KUKA KRL program: EPS_2_25999_MH2A_A_20251114084354.src

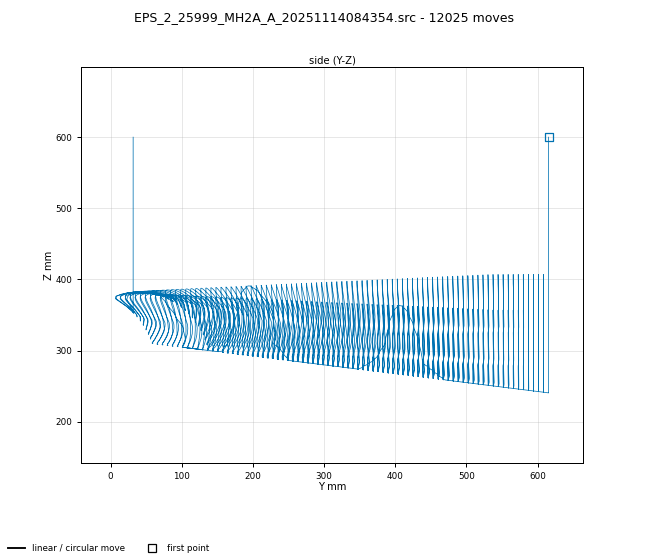
[picture p0: tool path of EPS_2_25999_MH2A_A_20251114084354.src, 12025 of 12027 moves have a stored position in this frame; points joined in program order, loops and branches not executed]
&ACCESS RVP
&REL 4
&COMMENT QRS 19112012
&PARAM EDITMASK = *
DEF PART()
EXT BAS (BAS_COMMAND :IN,REAL :IN )
INT I
BAS (#INITMOV,0 )

;KUKA QRS Post kuka4.cps  Date:22-06-2017 !

File_ID=2913

QRS_PRE_INIT()

;Init var - Until changes are made in qrs_pre_init
Outlet_Square_prg=0
Inlet_1_Square_prg=0
Inlet_2_Square_prg=0
Inlet_3_Square_prg=0
Inlet_4_Square_prg=0
Inlet_5_Square_prg=0

Outlet_1={X 0.000, Y 536.360, Z 332.000, B 0.000, E1 0.000 }
Inlet_1={X 0.000, Y 539.940, Z 282.000, B 0.000, E1 194.000 }
Outlet_1_type=150
Inlet_1_type=150
;QRS#1=Sidecore dimensions
;QRS#2=150-6" PVC SDR 28
;QRS#3=150-6" PVC SDR 28
;QRS#4=
;QRS#5=
;QRS#6=
;QRS#7=
;QRS#8=
;QRS#9=10-06 PSX
;QRS#10=10-06 PSX
;QRS#11=
;QRS#12=
;QRS#13=
;QRS#14=
;QRS#15=
;QRS#16=1220x127x686 2,25'
;QRS#17=EPS Height
;QRS#18=407
;QRS#19=*
;QRS#20= UPDATED VERSION 22-06-2017
;QRS#21=*
Outlet_Square=070
Inlet_1_Square=070
Inlet_2_Square=0
Inlet_3_Square=0
Inlet_4_Square=0
Inlet_5_Square=0
Mill_Square=1
Outlet_Square_Prg=203
Inlet_1_Square_prg=203

QRS_INIT()

$ADVANCE=5

; T1
PTP {E1 173.62,E2 173.62}
PTP {X 0,Y 615.486,A -85,B 0,C 180,E1 173.62,E2 173.62,E3 0,E4 0,E5 0,E6 0}
QRS_SPEED_INIT()
LIN {X 0,Y 615.486,Z 600,A -85,B 0,C 180,E1 173.62,E2 173.62,E3 0,E4 0,E5 0,E6 0} C_VEL
LIN {X 0,Y 615.486,Z 250.689,A -85,B 0,C 180,E1 173.62,E2 173.62} C_VEL
LIN {X 0,Y 615.486,Z 242.512,A -85,B 0,C 180,E1 173.62,E2 173.62} C_VEL
LIN {X 0,Y 615.477,Z 240.512,A -85,B 0,C 180,E1 173.434,E2 173.434} C_VEL
LIN {X 0,Y 615.498,Z 240.51,A -85,B 0,C 180,E1 170.803,E2 170.803} C_VEL
LIN {X 0,Y 615.487,Z 240.512,A -85,B 0,C 180,E1 168.141,E2 168.141} C_VEL
LIN {X 0,Y 615.477,Z 240.512,A -85,B 0,C 180,E1 165.452,E2 165.452} C_VEL
LIN {X 0,Y 615.487,Z 240.513,A -85,B 0,C 180,E1 162.731,E2 162.731} C_VEL
LIN {X 0,Y 615.49,Z 240.512,A -85,B 0,C 180,E1 159.969,E2 159.969} C_VEL
LIN {X 0,Y 615.493,Z 240.509,A -85,B 0,C 180,E1 157.157,E2 157.157} C_VEL
LIN {X 0,Y 615.478,Z 240.513,A -85,B 0,C 180,E1 154.434,E2 154.434} C_VEL
LIN {X 0,Y 615.479,Z 240.512,A -85,B 0,C 180,E1 152.086,E2 152.086} C_VEL
LIN {X 0,Y 615.49,Z 240.513,A -85,B 0,C 180,E1 149.842,E2 149.842} C_VEL
LIN {X 0,Y 615.495,Z 240.511,A -85,B 0,C 180,E1 147.545,E2 147.545} C_VEL
LIN {X 0,Y 615.487,Z 240.51,A -85,B 0,C 180,E1 145.187,E2 145.187} C_VEL
LIN {X 0,Y 615.487,Z 240.513,A -85,B 0,C 180,E1 142.76,E2 142.76} C_VEL
LIN {X 0,Y 615.479,Z 240.513,A -85,B 0,C 180,E1 139.913,E2 139.913} C_VEL
LIN {X 0,Y 615.5,Z 240.511,A -85,B 0,C 180,E1 137.651,E2 137.651} C_VEL
LIN {X 0,Y 615.477,Z 240.513,A -85,B 0,C 180,E1 134.933,E2 134.933} C_VEL
LIN {X 0,Y 615.49,Z 240.51,A -85,B 0,C 180,E1 132.083,E2 132.083} C_VEL
LIN {X 0,Y 615.491,Z 240.51,A -85,B 0,C 180,E1 129.751,E2 129.751} C_VEL
LIN {X 0,Y 615.476,Z 240.512,A -85,B 0,C 180,E1 126.939,E2 126.939} C_VEL
LIN {X 0,Y 615.481,Z 240.513,A -85,B 0,C 180,E1 124.704,E2 124.704} C_VEL
LIN {X 0,Y 615.498,Z 240.511,A -85,B 0,C 180,E1 122.336,E2 122.336} C_VEL
LIN {X 0,Y 615.49,Z 240.514,A -85,B 0,C 180,E1 119.407,E2 119.407} C_VEL
LIN {X 0,Y 615.492,Z 240.512,A -85,B 0,C 180,E1 116.445,E2 116.445} C_VEL
LIN {X 0,Y 615.483,Z 240.512,A -85,B 0,C 180,E1 113.557,E2 113.557} C_VEL
LIN {X 0,Y 615.485,Z 240.511,A -85,B 0,C 180,E1 110.732,E2 110.732} C_VEL
LIN {X 0,Y 615.492,Z 240.509,A -85,B 0,C 180,E1 108.613,E2 108.613} C_VEL
LIN {X 0,Y 615.483,Z 242.217,A -85,B 0,C 180,E1 107.271,E2 107.271} C_VEL
LIN {X 0,Y 615.491,Z 246.275,A -85,B 0,C 180,E1 104.55,E2 104.55} C_VEL
LIN {X 0,Y 615.487,Z 250.425,A -85,B 0,C 180,E1 101.862,E2 101.862} C_VEL
LIN {X 0,Y 615.47,Z 254.646,A -85,B 0,C 180,E1 99.2,E2 99.2} C_VEL
LIN {X 0,Y 615.491,Z 258.931,A -85,B 0,C 180,E1 96.557,E2 96.557} C_VEL
LIN {X 0,Y 615.464,Z 263.25,A -85,B 0,C 180,E1 93.929,E2 93.929} C_VEL
LIN {X 0,Y 615.465,Z 267.63,A -85,B 0,C 180,E1 91.309,E2 91.309} C_VEL
LIN {X 0,Y 615.493,Z 272.05,A -85,B 0,C 180,E1 88.692,E2 88.692} C_VEL
LIN {X 0,Y 615.433,Z 276.534,A -85,B 0,C 180,E1 86.072,E2 86.072} C_VEL
LIN {X 0,Y 615.492,Z 278.219,A -85,B 0,C 180,E1 85.088,E2 85.088} C_VEL
LIN {X 0,Y 615.471,Z 289.997,A -85,B 0,C 180,E1 84.76,E2 84.76} C_VEL
LIN {X 0,Y 615.441,Z 298.609,A -85,B 0,C 180,E1 84.431,E2 84.431} C_VEL
LIN {X 0,Y 615.429,Z 306.992,A -85,B 0,C 180,E1 84.02,E2 84.02} C_VEL
LIN {X 0,Y 615.456,Z 315.045,A -85,B 0,C 180,E1 83.526,E2 83.526} C_VEL
LIN {X 0,Y 615.498,Z 322.786,A -85,B 0,C 180,E1 82.944,E2 82.944} C_VEL
LIN {X 0,Y 615.496,Z 331.565,A -85,B 0,C 180,E1 82.125,E2 82.125} C_VEL
LIN {X 0,Y 615.497,Z 338.404,A -85,B 0,C 180,E1 81.299,E2 81.299} C_VEL
LIN {X 0,Y 615.495,Z 343.88,A -85,B 0,C 180,E1 80.471,E2 80.471} C_VEL
LIN {X 0,Y 615.49,Z 347.453,A -85,B 0,C 180,E1 79.807,E2 79.807} C_VEL
LIN {X 0,Y 615.492,Z 351.54,A -85,B 0,C 180,E1 78.808,E2 78.808} C_VEL
LIN {X 0,Y 615.491,Z 353.549,A -85,B 0,C 180,E1 78.14,E2 78.14} C_VEL
LIN {X 0,Y 615.496,Z 355.036,A -85,B 0,C 180,E1 77.471,E2 77.471} C_VEL
LIN {X 0,Y 615.491,Z 355.978,A -85,B 0,C 180,E1 76.8,E2 76.8} C_VEL
LIN {X 0,Y 615.491,Z 356.365,A -85,B 0,C 180,E1 76.056,E2 76.056} C_VEL
LIN {X 0,Y 615.493,Z 356.174,A -85,B 0,C 180,E1 75.452,E2 75.452} C_VEL
LIN {X 0,Y 615.491,Z 355.513,A -85,B 0,C 180,E1 74.775,E2 74.775} C_VEL
LIN {X 0,Y 615.491,Z 354.339,A -85,B 0,C 180,E1 74.096,E2 74.096} C_VEL
LIN {X 0,Y 615.492,Z 352.622,A -85,B 0,C 180,E1 73.415,E2 73.415} C_VEL
LIN {X 0,Y 615.496,Z 348.756,A -85,B 0,C 180,E1 72.388,E2 72.388} C_VEL
LIN {X 0,Y 615.496,Z 343.394,A -85,B 0,C 180,E1 71.355,E2 71.355} C_VEL
LIN {X 0,Y 615.498,Z 337.543,A -85,B 0,C 180,E1 70.49,E2 70.49} C_VEL
LIN {X 0,Y 615.496,Z 330.756,A -85,B 0,C 180,E1 69.702,E2 69.702} C_VEL
LIN {X 0,Y 615.497,Z 323.297,A -85,B 0,C 180,E1 69.008,E2 69.008} C_VEL
LIN {X 0,Y 615.471,Z 316.464,A -85,B 0,C 180,E1 68.481,E2 68.481} C_VEL
LIN {X 0,Y 615.468,Z 308.08,A -85,B 0,C 180,E1 67.952,E2 67.952} C_VEL
LIN {X 0,Y 615.494,Z 299.6,A -85,B 0,C 180,E1 67.525,E2 67.525} C_VEL
LIN {X 0,Y 615.487,Z 291.944,A -85,B 0,C 180,E1 67.218,E2 67.218} C_VEL
LIN {X 0,Y 615.496,Z 282.553,A -85,B 0,C 180,E1 66.935,E2 66.935} C_VEL
LIN {X 0,Y 615.485,Z 278.224,A -85,B 0,C 180,E1 66.823,E2 66.823} C_VEL
LIN {X 0,Y 615.458,Z 273.873,A -85,B 0,C 180,E1 64.284,E2 64.284} C_VEL
LIN {X 0,Y 615.494,Z 269.211,A -85,B 0,C 180,E1 61.544,E2 61.544} C_VEL
LIN {X 0,Y 615.444,Z 264.82,A -85,B 0,C 180,E1 58.916,E2 58.916} C_VEL
LIN {X 0,Y 615.444,Z 260.756,A -85,B 0,C 180,E1 56.468,E2 56.468} C_VEL
LIN {X 0,Y 615.462,Z 256.05,A -85,B 0,C 180,E1 53.575,E2 53.575} C_VEL
LIN {X 0,Y 615.42,Z 251.843,A -85,B 0,C 180,E1 50.942,E2 50.942} C_VEL
LIN {X 0,Y 615.456,Z 248.051,A -85,B 0,C 180,E1 48.525,E2 48.525} C_VEL
LIN {X 0,Y 615.495,Z 244.035,A -85,B 0,C 180,E1 45.853,E2 45.853} C_VEL
LIN {X 0,Y 615.491,Z 241.268,A -85,B 0,C 180,E1 44,E2 44} C_VEL
LIN {X 0,Y 615.457,Z 240.51,A -85,B 0,C 180,E1 43.046,E2 43.046} C_VEL
LIN {X 0,Y 615.484,Z 240.512,A -85,B 0,C 180,E1 40.604,E2 40.604} C_VEL
LIN {X 0,Y 615.473,Z 240.506,A -85,B 0,C 180,E1 38.012,E2 38.012} C_VEL
LIN {X 0,Y 615.489,Z 240.512,A -85,B 0,C 180,E1 35.613,E2 35.613} C_VEL
LIN {X 0,Y 615.446,Z 240.512,A -85,B 0,C 180,E1 33.237,E2 33.237} C_VEL
LIN {X 0,Y 615.491,Z 240.513,A -85,B 0,C 180,E1 30.917,E2 30.917} C_VEL
LIN {X 0,Y 615.481,Z 240.504,A -85,B 0,C 180,E1 28.452,E2 28.452} C_VEL
LIN {X 0,Y 615.454,Z 240.511,A -85,B 0,C 180,E1 25.715,E2 25.715} C_VEL
LIN {X 0,Y 615.488,Z 240.509,A -85,B 0,C 180,E1 22.843,E2 22.843} C_VEL
LIN {X 0,Y 615.484,Z 240.512,A -85,B 0,C 180,E1 20.031,E2 20.031} C_VEL
LIN {X 0,Y 615.472,Z 240.507,A -85,B 0,C 180,E1 17.269,E2 17.269} C_VEL
LIN {X 0,Y 615.448,Z 240.512,A -85,B 0,C 180,E1 14.548,E2 14.548} C_VEL
LIN {X 0,Y 615.49,Z 240.511,A -85,B 0,C 180,E1 11.859,E2 11.859} C_VEL
LIN {X 0,Y 615.498,Z 240.503,A -85,B 0,C 180,E1 9.197,E2 9.197} C_VEL
LIN {X 0,Y 615.443,Z 240.512,A -85,B 0,C 180,E1 6.554,E2 6.554} C_VEL
LIN {X 0,Y 615.491,Z 240.511,A -85,B 0,C 180,E1 3.927,E2 3.927} C_VEL
LIN {X 0,Y 615.494,Z 240.504,A -85,B 0,C 180,E1 1.307,E2 1.307} C_VEL
LIN {X 0,Y 615.445,Z 240.512,A -85,B 0,C 180,E1 -1.31,E2 -1.31} C_VEL
LIN {X 0,Y 615.489,Z 240.513,A -85,B 0,C 180,E1 -3.93,E2 -3.93} C_VEL
LIN {X 0,Y 615.489,Z 240.504,A -85,B 0,C 180,E1 -6.591,E2 -6.591} C_VEL
LIN {X 0,Y 615.446,Z 240.513,A -85,B 0,C 180,E1 -9.2,E2 -9.2} C_VEL
LIN {X 0,Y 615.49,Z 240.513,A -85,B 0,C 180,E1 -11.862,E2 -11.862} C_VEL
LIN {X 0,Y 615.483,Z 240.506,A -85,B 0,C 180,E1 -14.55,E2 -14.55} C_VEL
LIN {X 0,Y 615.451,Z 240.511,A -85,B 0,C 180,E1 -17.272,E2 -17.272} C_VEL
LIN {X 0,Y 615.485,Z 240.507,A -85,B 0,C 180,E1 -20.034,E2 -20.034} C_VEL
LIN {X 0,Y 615.487,Z 240.515,A -85,B 0,C 180,E1 -22.845,E2 -22.845} C_VEL
LIN {X 0,Y 615.492,Z 240.506,A -85,B 0,C 180,E1 -25.716,E2 -25.716} C_VEL
LIN {X 0,Y 615.452,Z 240.511,A -85,B 0,C 180,E1 -28.66,E2 -28.66} C_VEL
LIN {X 0,Y 615.486,Z 240.508,A -85,B 0,C 180,E1 -31.088,E2 -31.088} C_VEL
LIN {X 0,Y 615.495,Z 240.503,A -85,B 0,C 180,E1 -33.537,E2 -33.537} C_VEL
LIN {X 0,Y 615.442,Z 240.513,A -85,B 0,C 180,E1 -36.428,E2 -36.428} C_VEL
LIN {X 0,Y 615.489,Z 240.506,A -85,B 0,C 180,E1 -39.064,E2 -39.064} C_VEL
LIN {X 0,Y 615.491,Z 240.505,A -85,B 0,C 180,E1 -41.474,E2 -41.474} C_VEL
LIN {X 0,Y 615.443,Z 240.512,A -85,B 0,C 180,E1 -44.154,E2 -44.154} C_VEL
LIN {X 0,Y 615.492,Z 240.506,A -85,B 0,C 180,E1 -46.953,E2 -46.953} C_VEL
LIN {X 0,Y 615.489,Z 240.512,A -85,B 0,C 180,E1 -49.911,E2 -49.911} C_VEL
LIN {X 0,Y 615.473,Z 240.513,A -85,B 0,C 180,E1 -52.758,E2 -52.758} C_VEL
LIN {X 0,Y 615.474,Z 240.505,A -85,B 0,C 180,E1 -55.302,E2 -55.302} C_VEL
LIN {X 0,Y 615.486,Z 240.709,A -85,B 0,C 180,E1 -57.447,E2 -57.447} C_VEL
LIN {X 0,Y 615.494,Z 249.851,A -85,B 0,C 180,E1 -60.205,E2 -60.205} C_VEL
LIN {X 0,Y 615.493,Z 259.273,A -85,B 0,C 180,E1 -62.954,E2 -62.954} C_VEL
LIN {X 0,Y 615.447,Z 269.012,A -85,B 0,C 180,E1 -65.727,E2 -65.727} C_VEL
LIN {X 0,Y 615.453,Z 277.921,A -85,B 0,C 180,E1 -68.216,E2 -68.216} C_VEL
LIN {X 0,Y 615.447,Z 288.095,A -85,B 0,C 180,E1 -71.008,E2 -71.008} C_VEL
LIN {X 0,Y 615.45,Z 296.996,A -85,B 0,C 180,E1 -73.413,E2 -73.413} C_VEL
LIN {X 0,Y 615.489,Z 307.146,A -85,B 0,C 180,E1 -76.127,E2 -76.127} C_VEL
LIN {X 0,Y 615.476,Z 317.31,A -85,B 0,C 180,E1 -78.808,E2 -78.808} C_VEL
LIN {X 0,Y 615.485,Z 324.917,A -85,B 0,C 180,E1 -80.802,E2 -80.802} C_VEL
LIN {X 0,Y 615.492,Z 338.188,A -85,B 0,C 180,E1 -81.133,E2 -81.133} C_VEL
LIN {X 0,Y 615.472,Z 347.248,A -85,B 0,C 180,E1 -81.464,E2 -81.464} C_VEL
LIN {X 0,Y 615.475,Z 355.931,A -85,B 0,C 180,E1 -81.877,E2 -81.877} C_VEL
LIN {X 0,Y 615.492,Z 364.211,A -85,B 0,C 180,E1 -82.373,E2 -82.373} C_VEL
LIN {X 0,Y 615.499,Z 371.943,A -85,B 0,C 180,E1 -82.943,E2 -82.943} C_VEL
LIN {X 0,Y 615.498,Z 377.655,A -85,B 0,C 180,E1 -83.444,E2 -83.444} C_VEL
LIN {X 0,Y 615.5,Z 383.929,A -85,B 0,C 180,E1 -84.102,E2 -84.102} C_VEL
LIN {X 0,Y 615.495,Z 389.142,A -85,B 0,C 180,E1 -84.76,E2 -84.76} C_VEL
LIN {X 0,Y 615.495,Z 393.487,A -85,B 0,C 180,E1 -85.416,E2 -85.416} C_VEL
LIN {X 0,Y 615.491,Z 398.607,A -85,B 0,C 180,E1 -86.4,E2 -86.4} C_VEL
LIN {X 0,Y 615.488,Z 401.224,A -85,B 0,C 180,E1 -87.056,E2 -87.056} C_VEL
LIN {X 0,Y 615.499,Z 404.087,A -85,B 0,C 180,E1 -88.038,E2 -88.038} C_VEL
LIN {X 0,Y 615.493,Z 405.331,A -85,B 0,C 180,E1 -88.692,E2 -88.692} C_VEL
LIN {X 0,Y 615.491,Z 406.105,A -85,B 0,C 180,E1 -89.347,E2 -89.347} C_VEL
LIN {X 0,Y 615.491,Z 406.389,A -85,B 0,C 180,E1 -90.001,E2 -90.001} C_VEL
LIN {X 0,Y 615.491,Z 406.104,A -85,B 0,C 180,E1 -90.655,E2 -90.655} C_VEL
LIN {X 0,Y 615.493,Z 405.329,A -85,B 0,C 180,E1 -91.309,E2 -91.309} C_VEL
LIN {X 0,Y 615.499,Z 404.083,A -85,B 0,C 180,E1 -91.964,E2 -91.964} C_VEL
LIN {X 0,Y 615.488,Z 401.218,A -85,B 0,C 180,E1 -92.946,E2 -92.946} C_VEL
LIN {X 0,Y 615.491,Z 398.6,A -85,B 0,C 180,E1 -93.601,E2 -93.601} C_VEL
LIN {X 0,Y 615.495,Z 393.478,A -85,B 0,C 180,E1 -94.585,E2 -94.585} C_VEL
LIN {X 0,Y 615.495,Z 387.962,A -85,B 0,C 180,E1 -95.406,E2 -95.406} C_VEL
LIN {X 0,Y 615.498,Z 381.01,A -85,B 0,C 180,E1 -96.228,E2 -96.228} C_VEL
LIN {X 0,Y 615.498,Z 373.855,A -85,B 0,C 180,E1 -96.901,E2 -96.901} C_VEL
LIN {X 0,Y 615.489,Z 366.61,A -85,B 0,C 180,E1 -97.464,E2 -97.464} C_VEL
LIN {X 0,Y 615.483,Z 358.857,A -85,B 0,C 180,E1 -97.959,E2 -97.959} C_VEL
LIN {X 0,Y 615.469,Z 350.903,A -85,B 0,C 180,E1 -98.372,E2 -98.372} C_VEL
LIN {X 0,Y 615.482,Z 341.736,A -85,B 0,C 180,E1 -98.744,E2 -98.744} C_VEL
LIN {X 0,Y 615.493,Z 333.661,A -85,B 0,C 180,E1 -98.992,E2 -98.992} C_VEL
LIN {X 0,Y 615.485,Z 324.911,A -85,B 0,C 180,E1 -99.2,E2 -99.2} C_VEL
LIN {X 0,Y 615.49,Z 314.759,A -85,B 0,C 180,E1 -101.862,E2 -101.862} C_VEL
LIN {X 0,Y 615.469,Z 304.605,A -85,B 0,C 180,E1 -104.55,E2 -104.55} C_VEL
LIN {X 0,Y 615.472,Z 294.44,A -85,B 0,C 180,E1 -107.272,E2 -107.272} C_VEL
LIN {X 0,Y 615.442,Z 284.276,A -85,B 0,C 180,E1 -110.035,E2 -110.035} C_VEL
LIN {X 0,Y 615.433,Z 275.946,A -85,B 0,C 180,E1 -112.333,E2 -112.333} C_VEL
LIN {X 0,Y 615.495,Z 266.454,A -85,B 0,C 180,E1 -114.992,E2 -114.992} C_VEL
LIN {X 0,Y 615.475,Z 257.545,A -85,B 0,C 180,E1 -117.547,E2 -117.547} C_VEL
LIN {X 0,Y 615.488,Z 248.618,A -85,B 0,C 180,E1 -120.161,E2 -120.161} C_VEL
LIN {X 0,Y 615.485,Z 240.511,A -85,B 0,C 180,E1 -122.652,E2 -122.652} C_VEL
LIN {X 0,Y 615.485,Z 240.511,A -85,B 0,C 180,E1 -124.816,E2 -124.816} C_VEL
LIN {X 0,Y 615.492,Z 240.513,A -85,B 0,C 180,E1 -127.243,E2 -127.243} C_VEL
LIN {X 0,Y 615.48,Z 240.513,A -85,B 0,C 180,E1 -130.088,E2 -130.088} C_VEL
LIN {X 0,Y 615.496,Z 240.513,A -85,B 0,C 180,E1 -132.353,E2 -132.353} C_VEL
LIN {X 0,Y 615.49,Z 240.51,A -85,B 0,C 180,E1 -135.069,E2 -135.069} C_VEL
LIN {X 0,Y 615.476,Z 240.512,A -85,B 0,C 180,E1 -137.922,E2 -137.922} C_VEL
LIN {X 0,Y 615.483,Z 240.512,A -85,B 0,C 180,E1 -140.249,E2 -140.249} C_VEL
LIN {X 0,Y 615.478,Z 240.512,A -85,B 0,C 180,E1 -143.065,E2 -143.065} C_VEL
LIN {X 0,Y 615.48,Z 240.513,A -85,B 0,C 180,E1 -145.301,E2 -145.301} C_VEL
LIN {X 0,Y 615.492,Z 240.512,A -85,B 0,C 180,E1 -147.669,E2 -147.669} C_VEL
LIN {X 0,Y 615.494,Z 240.514,A -85,B 0,C 180,E1 -150.593,E2 -150.593} C_VEL
LIN {X 0,Y 615.477,Z 240.513,A -85,B 0,C 180,E1 -152.958,E2 -152.958} C_VEL
LIN {X 0,Y 615.494,Z 240.513,A -85,B 0,C 180,E1 -155.727,E2 -155.727} C_VEL
LIN {X 0,Y 615.494,Z 240.512,A -85,B 0,C 180,E1 -158.568,E2 -158.568} C_VEL
LIN {X 0,Y 615.479,Z 240.512,A -85,B 0,C 180,E1 -161.399,E2 -161.399} C_VEL
LIN {X 0,Y 615.491,Z 240.51,A -85,B 0,C 180,E1 -164.094,E2 -164.094} C_VEL
LIN {X 0,Y 615.497,Z 240.513,A -85,B 0,C 180,E1 -166.798,E2 -166.798} C_VEL
LIN {X 0,Y 615.477,Z 240.513,A -85,B 0,C 180,E1 -169.472,E2 -169.472} C_VEL
LIN {X 0,Y 615.481,Z 240.512,A -85,B 0,C 180,E1 -172.123,E2 -172.123} C_VEL
LIN {X 0,Y 615.487,Z 240.513,A -85,B 0,C 180,E1 -174.758,E2 -174.758} C_VEL
LIN {X 0,Y 615.491,Z 240.509,A -85,B 0,C 180,E1 -177.381,E2 -177.381} C_VEL
LIN {X 0,Y 615.489,Z 240.514,A -85,B 0,C 180,E1 -179.999,E2 -179.999} C_VEL
LIN {X 0,Y 615.479,Z 240.512,A -85,B 0,C 180,E1 -182.617,E2 -182.617} C_VEL
LIN {X 0,Y 615.497,Z 240.509,A -85,B 0,C 180,E1 -185.24,E2 -185.24} C_VEL
LIN {X 0,Y 615.477,Z 240.512,A -85,B 0,C 180,E1 -186.566,E2 -186.566} C_VEL
LIN {X 0,Y 614.814,Z 240.657,A -85,B 0,C 180,E1 -187.112,E2 -187.112} C_VEL
LIN {X 0,Y 611.991,Z 241.07,A -85,B 0,C 180,E1 -187.998,E2 -187.998} C_VEL
LIN {X 0,Y 609.6,Z 241.378,A -85,B 0,C 180,E1 -188.711,E2 -188.711} C_VEL
LIN {X 0,Y 608.56,Z 241.496,A -85,B 0,C 180,E1 -189.26,E2 -189.26} C_VEL
LIN {X 0,Y 608.468,Z 241.506,A -85,B 0,C 180,E1 -189.447,E2 -189.447} C_VEL
LIN {X 0,Y 608.461,Z 241.509,A -85,B 0,C 180,E1 -191.998,E2 -191.998} C_VEL
LIN {X 0,Y 608.47,Z 241.506,A -85,B 0,C 180,E1 -194.719,E2 -194.719} C_VEL
LIN {X 0,Y 608.453,Z 241.508,A -85,B 0,C 180,E1 -197.475,E2 -197.475} C_VEL
LIN {X 0,Y 608.463,Z 241.508,A -85,B 0,C 180,E1 -200.272,E2 -200.272} C_VEL
LIN {X 0,Y 608.451,Z 241.51,A -85,B 0,C 180,E1 -203.122,E2 -203.122} C_VEL
LIN {X 0,Y 608.463,Z 241.507,A -85,B 0,C 180,E1 -205.718,E2 -205.718} C_VEL
LIN {X 0,Y 608.452,Z 241.511,A -85,B 0,C 180,E1 -208.265,E2 -208.265} C_VEL
LIN {X 0,Y 608.474,Z 241.506,A -85,B 0,C 180,E1 -210.542,E2 -210.542} C_VEL
LIN {X 0,Y 608.462,Z 241.507,A -85,B 0,C 180,E1 -212.877,E2 -212.877} C_VEL
LIN {X 0,Y 608.44,Z 241.512,A -85,B 0,C 180,E1 -215.276,E2 -215.276} C_VEL
LIN {X 0,Y 608.464,Z 241.507,A -85,B 0,C 180,E1 -217.744,E2 -217.744} C_VEL
LIN {X 0,Y 608.447,Z 241.511,A -85,B 0,C 180,E1 -220.328,E2 -220.328} C_VEL
LIN {X 0,Y 608.447,Z 241.509,A -85,B 0,C 180,E1 -222.958,E2 -222.958} C_VEL
LIN {X 0,Y 608.453,Z 241.508,A -85,B 0,C 180,E1 -225.734,E2 -225.734} C_VEL
LIN {X 0,Y 608.462,Z 241.508,A -85,B 0,C 180,E1 -228.655,E2 -228.655} C_VEL
LIN {X 0,Y 608.464,Z 241.508,A -85,B 0,C 180,E1 -231.411,E2 -231.411} C_VEL
LIN {X 0,Y 608.471,Z 241.506,A -85,B 0,C 180,E1 -233.948,E2 -233.948} C_VEL
LIN {X 0,Y 608.472,Z 241.506,A -85,B 0,C 180,E1 -236.329,E2 -236.329} C_VEL
LIN {X 0,Y 608.466,Z 241.508,A -85,B 0,C 180,E1 -238.725,E2 -238.725} C_VEL
LIN {X 0,Y 608.471,Z 241.506,A -85,B 0,C 180,E1 -241.376,E2 -241.376} C_VEL
LIN {X 0,Y 608.444,Z 241.509,A -85,B 0,C 180,E1 -243.964,E2 -243.964} C_VEL
LIN {X 0,Y 608.461,Z 241.507,A -85,B 0,C 180,E1 -246.154,E2 -246.154} C_VEL
LIN {X 0,Y 608.468,Z 241.506,A -85,B 0,C 180,E1 -248.308,E2 -248.308} C_VEL
LIN {X 0,Y 608.467,Z 241.506,A -85,B 0,C 180,E1 -251.278,E2 -251.278} C_VEL
LIN {X 0,Y 608.442,Z 241.748,A -85,B 0,C 180,E1 -251.827,E2 -251.827} C_VEL
LIN {X 0,Y 608.45,Z 245.854,A -85,B 0,C 180,E1 -254.593,E2 -254.593} C_VEL
LIN {X 0,Y 608.451,Z 249.952,A -85,B 0,C 180,E1 -257.322,E2 -257.322} C_VEL
LIN {X 0,Y 608.44,Z 254.187,A -85,B 0,C 180,E1 -260.022,E2 -260.022} C_VEL
LIN {X 0,Y 608.43,Z 258.477,A -85,B 0,C 180,E1 -262.699,E2 -262.699} C_VEL
LIN {X 0,Y 608.455,Z 262.818,A -85,B 0,C 180,E1 -265.362,E2 -265.362} C_VEL
LIN {X 0,Y 608.404,Z 267.215,A -85,B 0,C 180,E1 -268.013,E2 -268.013} C_VEL
LIN {X 0,Y 608.407,Z 271.661,A -85,B 0,C 180,E1 -270.661,E2 -270.661} C_VEL
LIN {X 0,Y 608.41,Z 276.158,A -85,B 0,C 180,E1 -273.31,E2 -273.31} C_VEL
LIN {X 0,Y 608.414,Z 278.71,A -85,B 0,C 180,E1 -274.803,E2 -274.803} C_VEL
LIN {X 0,Y 608.465,Z 290.221,A -85,B 0,C 180,E1 -275.135,E2 -275.135} C_VEL
LIN {X 0,Y 608.452,Z 298.827,A -85,B 0,C 180,E1 -275.467,E2 -275.467} C_VEL
LIN {X 0,Y 608.416,Z 307.241,A -85,B 0,C 180,E1 -275.883,E2 -275.883} C_VEL
LIN {X 0,Y 608.435,Z 314.894,A -85,B 0,C 180,E1 -276.352,E2 -276.352} C_VEL
LIN {X 0,Y 608.467,Z 322.027,A -85,B 0,C 180,E1 -276.882,E2 -276.882} C_VEL
LIN {X 0,Y 608.464,Z 328.587,A -85,B 0,C 180,E1 -277.465,E2 -277.465} C_VEL
LIN {X 0,Y 608.458,Z 334.831,A -85,B 0,C 180,E1 -278.133,E2 -278.133} C_VEL
LIN {X 0,Y 608.448,Z 340.029,A -85,B 0,C 180,E1 -278.803,E2 -278.803} C_VEL
LIN {X 0,Y 608.432,Z 343.398,A -85,B 0,C 180,E1 -279.305,E2 -279.305} C_VEL
LIN {X 0,Y 608.433,Z 347.195,A -85,B 0,C 180,E1 -279.977,E2 -279.977} C_VEL
LIN {X 0,Y 608.424,Z 351.373,A -85,B 0,C 180,E1 -280.946,E2 -280.946} C_VEL
LIN {X 0,Y 608.434,Z 354.534,A -85,B 0,C 180,E1 -281.999,E2 -281.999} C_VEL
LIN {X 0,Y 608.416,Z 355.871,A -85,B 0,C 180,E1 -282.677,E2 -282.677} C_VEL
LIN {X 0,Y 608.433,Z 356.701,A -85,B 0,C 180,E1 -283.356,E2 -283.356} C_VEL
LIN {X 0,Y 608.419,Z 357,A -85,B 0,C 180,E1 -284.038,E2 -284.038} C_VEL
LIN {X 0,Y 608.42,Z 356.707,A -85,B 0,C 180,E1 -284.721,E2 -284.721} C_VEL
LIN {X 0,Y 608.416,Z 355.88,A -85,B 0,C 180,E1 -285.406,E2 -285.406} C_VEL
LIN {X 0,Y 608.447,Z 353.454,A -85,B 0,C 180,E1 -286.531,E2 -286.531} C_VEL
LIN {X 0,Y 608.428,Z 350.112,A -85,B 0,C 180,E1 -287.476,E2 -287.476} C_VEL
LIN {X 0,Y 608.443,Z 345.378,A -85,B 0,C 180,E1 -288.441,E2 -288.441} C_VEL
LIN {X 0,Y 608.464,Z 340.518,A -85,B 0,C 180,E1 -289.218,E2 -289.218} C_VEL
LIN {X 0,Y 608.463,Z 335.138,A -85,B 0,C 180,E1 -289.921,E2 -289.921} C_VEL
LIN {X 0,Y 608.46,Z 329.413,A -85,B 0,C 180,E1 -290.544,E2 -290.544} C_VEL
LIN {X 0,Y 608.47,Z 322.648,A -85,B 0,C 180,E1 -291.157,E2 -291.157} C_VEL
LIN {X 0,Y 608.457,Z 315.575,A -85,B 0,C 180,E1 -291.691,E2 -291.691} C_VEL
LIN {X 0,Y 608.45,Z 308.474,A -85,B 0,C 180,E1 -292.137,E2 -292.137} C_VEL
LIN {X 0,Y 608.503,Z 299.706,A -85,B 0,C 180,E1 -292.582,E2 -292.582} C_VEL
LIN {X 0,Y 608.48,Z 290.597,A -85,B 0,C 180,E1 -292.942,E2 -292.942} C_VEL
LIN {X 0,Y 608.495,Z 281.297,A -85,B 0,C 180,E1 -293.211,E2 -293.211} C_VEL
LIN {X 0,Y 608.426,Z 278.72,A -85,B 0,C 180,E1 -293.281,E2 -293.281} C_VEL
LIN {X 0,Y 608.399,Z 274.019,A -85,B 0,C 180,E1 -296.036,E2 -296.036} C_VEL
LIN {X 0,Y 608.424,Z 269.66,A -85,B 0,C 180,E1 -298.616,E2 -298.616} C_VEL
LIN {X 0,Y 608.386,Z 265.243,A -85,B 0,C 180,E1 -301.262,E2 -301.262} C_VEL
LIN {X 0,Y 608.398,Z 261.182,A -85,B 0,C 180,E1 -303.728,E2 -303.728} C_VEL
LIN {X 0,Y 608.426,Z 257.346,A -85,B 0,C 180,E1 -306.092,E2 -306.092} C_VEL
LIN {X 0,Y 608.393,Z 253.362,A -85,B 0,C 180,E1 -308.592,E2 -308.592} C_VEL
LIN {X 0,Y 608.387,Z 249.076,A -85,B 0,C 180,E1 -311.337,E2 -311.337} C_VEL
LIN {X 0,Y 608.436,Z 245.279,A -85,B 0,C 180,E1 -313.871,E2 -313.871} C_VEL
LIN {X 0,Y 608.427,Z 241.958,A -85,B 0,C 180,E1 -316.13,E2 -316.13} C_VEL
LIN {X 0,Y 608.428,Z 241.507,A -85,B 0,C 180,E1 -317.041,E2 -317.041} C_VEL
LIN {X 0,Y 608.44,Z 241.51,A -85,B 0,C 180,E1 -319.698,E2 -319.698} C_VEL
LIN {X 0,Y 608.46,Z 241.504,A -85,B 0,C 180,E1 -322.256,E2 -322.256} C_VEL
LIN {X 0,Y 608.467,Z 241.502,A -85,B 0,C 180,E1 -325.09,E2 -325.09} C_VEL
LIN {X 0,Y 608.443,Z 241.506,A -85,B 0,C 180,E1 -327.906,E2 -327.906} C_VEL
LIN {X 0,Y 608.451,Z 241.506,A -85,B 0,C 180,E1 -330.222,E2 -330.222} C_VEL
LIN {X 0,Y 608.465,Z 241.503,A -85,B 0,C 180,E1 -332.792,E2 -332.792} C_VEL
LIN {X 0,Y 608.435,Z 241.512,A -85,B 0,C 180,E1 -335.43,E2 -335.43} C_VEL
LIN {X 0,Y 608.462,Z 241.506,A -85,B 0,C 180,E1 -338.31,E2 -338.31} C_VEL
LIN {X 0,Y 608.466,Z 241.504,A -85,B 0,C 180,E1 -341.281,E2 -341.281} C_VEL
LIN {X 0,Y 608.426,Z 241.507,A -85,B 0,C 180,E1 -343.907,E2 -343.907} C_VEL
LIN {X 0,Y 608.463,Z 241.506,A -85,B 0,C 180,E1 -346.645,E2 -346.645} C_VEL
LIN {X 0,Y 608.467,Z 241.505,A -85,B 0,C 180,E1 -349.352,E2 -349.352} C_VEL
LIN {X 0,Y 608.419,Z 241.508,A -85,B 0,C 180,E1 -352.034,E2 -352.034} C_VEL
LIN {X 0,Y 608.464,Z 241.505,A -85,B 0,C 180,E1 -354.699,E2 -354.699} C_VEL
LIN {X 0,Y 608.479,Z 241.505,A -85,B 0,C 180,E1 -357.353,E2 -357.353} C_VEL
LIN {X 0,Y 608.452,Z 241.504,A -85,B 0,C 180,E1 -360.001,E2 -360.001} C_VEL
LIN {X 0,Y 608.468,Z 241.504,A -85,B 0,C 180,E1 -362.649,E2 -362.649} C_VEL
LIN {X 0,Y 608.462,Z 241.507,A -85,B 0,C 180,E1 -365.303,E2 -365.303} C_VEL
LIN {X 0,Y 608.463,Z 241.503,A -85,B 0,C 180,E1 -367.968,E2 -367.968} C_VEL
LIN {X 0,Y 608.439,Z 241.505,A -85,B 0,C 180,E1 -370.948,E2 -370.948} C_VEL
LIN {X 0,Y 608.462,Z 241.51,A -85,B 0,C 180,E1 -373.357,E2 -373.357} C_VEL
LIN {X 0,Y 608.461,Z 241.504,A -85,B 0,C 180,E1 -376.095,E2 -376.095} C_VEL
LIN {X 0,Y 608.431,Z 241.506,A -85,B 0,C 180,E1 -378.871,E2 -378.871} C_VEL
LIN {X 0,Y 608.471,Z 241.503,A -85,B 0,C 180,E1 -381.692,E2 -381.692} C_VEL
LIN {X 0,Y 608.446,Z 241.51,A -85,B 0,C 180,E1 -384.572,E2 -384.572} C_VEL
LIN {X 0,Y 608.449,Z 241.506,A -85,B 0,C 180,E1 -387.205,E2 -387.205} C_VEL
LIN {X 0,Y 608.463,Z 241.503,A -85,B 0,C 180,E1 -389.973,E2 -389.973} C_VEL
LIN {X 0,Y 608.465,Z 241.507,A -85,B 0,C 180,E1 -392.525,E2 -392.525} C_VEL
LIN {X 0,Y 608.413,Z 241.509,A -85,B 0,C 180,E1 -394.903,E2 -394.903} C_VEL
LIN {X 0,Y 608.459,Z 241.503,A -85,B 0,C 180,E1 -397.748,E2 -397.748} C_VEL
LIN {X 0,Y 608.449,Z 241.511,A -85,B 0,C 180,E1 -400.331,E2 -400.331} C_VEL
LIN {X 0,Y 608.478,Z 241.505,A -85,B 0,C 180,E1 -403.311,E2 -403.311} C_VEL
LIN {X 0,Y 608.446,Z 241.506,A -85,B 0,C 180,E1 -406.13,E2 -406.13} C_VEL
LIN {X 0,Y 608.454,Z 241.504,A -85,B 0,C 180,E1 -408.825,E2 -408.825} C_VEL
LIN {X 0,Y 608.439,Z 241.508,A -85,B 0,C 180,E1 -411.764,E2 -411.764} C_VEL
LIN {X 0,Y 608.432,Z 241.507,A -85,B 0,C 180,E1 -413.957,E2 -413.957} C_VEL
LIN {X 0,Y 608.462,Z 241.508,A -85,B 0,C 180,E1 -416.331,E2 -416.331} C_VEL
LIN {X 0,Y 608.502,Z 241.714,A -85,B 0,C 180,E1 -417.334,E2 -417.334} C_VEL
LIN {X 0,Y 608.514,Z 248.607,A -85,B 0,C 180,E1 -419.459,E2 -419.459} C_VEL
LIN {X 0,Y 608.481,Z 257.608,A -85,B 0,C 180,E1 -422.111,E2 -422.111} C_VEL
LIN {X 0,Y 608.478,Z 266.549,A -85,B 0,C 180,E1 -424.701,E2 -424.701} C_VEL
LIN {X 0,Y 608.426,Z 276.545,A -85,B 0,C 180,E1 -427.532,E2 -427.532} C_VEL
LIN {X 0,Y 608.42,Z 285.709,A -85,B 0,C 180,E1 -430.078,E2 -430.078} C_VEL
LIN {X 0,Y 608.426,Z 295.927,A -85,B 0,C 180,E1 -432.87,E2 -432.87} C_VEL
LIN {X 0,Y 608.459,Z 306.146,A -85,B 0,C 180,E1 -435.622,E2 -435.622} C_VEL
LIN {X 0,Y 608.431,Z 316.365,A -85,B 0,C 180,E1 -438.339,E2 -438.339} C_VEL
LIN {X 0,Y 608.425,Z 325.306,A -85,B 0,C 180,E1 -440.694,E2 -440.694} C_VEL
LIN {X 0,Y 608.498,Z 338.509,A -85,B 0,C 180,E1 -441.031,E2 -441.031} C_VEL
LIN {X 0,Y 608.472,Z 347.555,A -85,B 0,C 180,E1 -441.365,E2 -441.365} C_VEL
LIN {X 0,Y 608.456,Z 356.249,A -85,B 0,C 180,E1 -441.783,E2 -441.783} C_VEL
LIN {X 0,Y 608.47,Z 364.555,A -85,B 0,C 180,E1 -442.284,E2 -442.284} C_VEL
LIN {X 0,Y 608.464,Z 372.412,A -85,B 0,C 180,E1 -442.868,E2 -442.868} C_VEL
LIN {X 0,Y 608.466,Z 379.364,A -85,B 0,C 180,E1 -443.496,E2 -443.496} C_VEL
LIN {X 0,Y 608.47,Z 387.198,A -85,B 0,C 180,E1 -444.367,E2 -444.367} C_VEL
LIN {X 0,Y 608.448,Z 393.032,A -85,B 0,C 180,E1 -445.197,E2 -445.197} C_VEL
LIN {X 0,Y 608.434,Z 397.635,A -85,B 0,C 180,E1 -446.027,E2 -446.027} C_VEL
LIN {X 0,Y 608.424,Z 400.625,A -85,B 0,C 180,E1 -446.69,E2 -446.69} C_VEL
LIN {X 0,Y 608.423,Z 402.934,A -85,B 0,C 180,E1 -447.353,E2 -447.353} C_VEL
LIN {X 0,Y 608.444,Z 404.68,A -85,B 0,C 180,E1 -448.015,E2 -448.015} C_VEL
LIN {X 0,Y 608.446,Z 405.935,A -85,B 0,C 180,E1 -448.677,E2 -448.677} C_VEL
LIN {X 0,Y 608.434,Z 406.714,A -85,B 0,C 180,E1 -449.339,E2 -449.339} C_VEL
LIN {X 0,Y 608.431,Z 407,A -85,B 0,C 180,E1 -450.001,E2 -450.001} C_VEL
LIN {X 0,Y 608.434,Z 406.713,A -85,B 0,C 180,E1 -450.663,E2 -450.663} C_VEL
LIN {X 0,Y 608.445,Z 405.932,A -85,B 0,C 180,E1 -451.325,E2 -451.325} C_VEL
LIN {X 0,Y 608.444,Z 404.676,A -85,B 0,C 180,E1 -451.987,E2 -451.987} C_VEL
LIN {X 0,Y 608.444,Z 401.783,A -85,B 0,C 180,E1 -452.98,E2 -452.98} C_VEL
LIN {X 0,Y 608.445,Z 399.142,A -85,B 0,C 180,E1 -453.643,E2 -453.643} C_VEL
LIN {X 0,Y 608.431,Z 393.98,A -85,B 0,C 180,E1 -454.639,E2 -454.639} C_VEL
LIN {X 0,Y 608.46,Z 388.424,A -85,B 0,C 180,E1 -455.469,E2 -455.469} C_VEL
LIN {X 0,Y 608.455,Z 380.674,A -85,B 0,C 180,E1 -456.375,E2 -456.375} C_VEL
LIN {X 0,Y 608.456,Z 373.405,A -85,B 0,C 180,E1 -457.05,E2 -457.05} C_VEL
LIN {X 0,Y 608.471,Z 365.748,A -85,B 0,C 180,E1 -457.634,E2 -457.634} C_VEL
LIN {X 0,Y 608.477,Z 357.705,A -85,B 0,C 180,E1 -458.135,E2 -458.135} C_VEL
LIN {X 0,Y 608.478,Z 349.371,A -85,B 0,C 180,E1 -458.553,E2 -458.553} C_VEL
LIN {X 0,Y 608.485,Z 340.865,A -85,B 0,C 180,E1 -458.887,E2 -458.887} C_VEL
LIN {X 0,Y 608.506,Z 331.552,A -85,B 0,C 180,E1 -459.159,E2 -459.159} C_VEL
LIN {X 0,Y 608.424,Z 325.299,A -85,B 0,C 180,E1 -459.307,E2 -459.307} C_VEL
LIN {X 0,Y 608.433,Z 315.081,A -85,B 0,C 180,E1 -462.001,E2 -462.001} C_VEL
LIN {X 0,Y 608.428,Z 304.862,A -85,B 0,C 180,E1 -464.722,E2 -464.722} C_VEL
LIN {X 0,Y 608.461,Z 294.643,A -85,B 0,C 180,E1 -467.477,E2 -467.477} C_VEL
LIN {X 0,Y 608.415,Z 284.425,A -85,B 0,C 180,E1 -470.277,E2 -470.277} C_VEL
LIN {X 0,Y 608.437,Z 275.485,A -85,B 0,C 180,E1 -472.766,E2 -472.766} C_VEL
LIN {X 0,Y 608.478,Z 266.542,A -85,B 0,C 180,E1 -475.301,E2 -475.301} C_VEL
LIN {X 0,Y 608.482,Z 257.601,A -85,B 0,C 180,E1 -477.891,E2 -477.891} C_VEL
LIN {X 0,Y 608.515,Z 248.637,A -85,B 0,C 180,E1 -480.543,E2 -480.543} C_VEL
LIN {X 0,Y 608.466,Z 241.507,A -85,B 0,C 180,E1 -482.774,E2 -482.774} C_VEL
LIN {X 0,Y 608.44,Z 241.512,A -85,B 0,C 180,E1 -485.279,E2 -485.279} C_VEL
LIN {X 0,Y 608.468,Z 241.506,A -85,B 0,C 180,E1 -487.747,E2 -487.747} C_VEL
LIN {X 0,Y 608.451,Z 241.511,A -85,B 0,C 180,E1 -490.328,E2 -490.328} C_VEL
LIN {X 0,Y 608.481,Z 241.506,A -85,B 0,C 180,E1 -493.309,E2 -493.309} C_VEL
LIN {X 0,Y 608.464,Z 241.507,A -85,B 0,C 180,E1 -496.13,E2 -496.13} C_VEL
LIN {X 0,Y 608.457,Z 241.508,A -85,B 0,C 180,E1 -498.823,E2 -498.823} C_VEL
LIN {X 0,Y 608.459,Z 241.508,A -85,B 0,C 180,E1 -501.761,E2 -501.761} C_VEL
LIN {X 0,Y 608.45,Z 241.508,A -85,B 0,C 180,E1 -503.955,E2 -503.955} C_VEL
LIN {X 0,Y 608.474,Z 241.506,A -85,B 0,C 180,E1 -506.329,E2 -506.329} C_VEL
LIN {X 0,Y 608.451,Z 241.51,A -85,B 0,C 180,E1 -508.733,E2 -508.733} C_VEL
LIN {X 0,Y 608.475,Z 241.506,A -85,B 0,C 180,E1 -511.381,E2 -511.381} C_VEL
LIN {X 0,Y 608.482,Z 241.505,A -85,B 0,C 180,E1 -514.278,E2 -514.278} C_VEL
LIN {X 0,Y 608.448,Z 241.51,A -85,B 0,C 180,E1 -516.875,E2 -516.875} C_VEL
LIN {X 0,Y 608.465,Z 241.507,A -85,B 0,C 180,E1 -519.323,E2 -519.323} C_VEL
LIN {X 0,Y 608.452,Z 241.51,A -85,B 0,C 180,E1 -521.827,E2 -521.827} C_VEL
LIN {X 0,Y 608.475,Z 241.506,A -85,B 0,C 180,E1 -524.593,E2 -524.593} C_VEL
LIN {X 0,Y 608.473,Z 241.505,A -85,B 0,C 180,E1 -527.322,E2 -527.322} C_VEL
LIN {X 0,Y 608.45,Z 241.509,A -85,B 0,C 180,E1 -530.022,E2 -530.022} C_VEL
LIN {X 0,Y 608.467,Z 241.508,A -85,B 0,C 180,E1 -532.7,E2 -532.7} C_VEL
LIN {X 0,Y 608.457,Z 241.507,A -85,B 0,C 180,E1 -535.361,E2 -535.361} C_VEL
LIN {X 0,Y 608.459,Z 241.509,A -85,B 0,C 180,E1 -538.013,E2 -538.013} C_VEL
LIN {X 0,Y 608.476,Z 241.506,A -85,B 0,C 180,E1 -540.661,E2 -540.661} C_VEL
LIN {X 0,Y 608.487,Z 241.504,A -85,B 0,C 180,E1 -543.309,E2 -543.309} C_VEL
LIN {X 0,Y 608.466,Z 241.509,A -85,B 0,C 180,E1 -545.966,E2 -545.966} C_VEL
LIN {X 0,Y 608.45,Z 241.508,A -85,B 0,C 180,E1 -548.635,E2 -548.635} C_VEL
LIN {X 0,Y 608.468,Z 241.506,A -85,B 0,C 180,E1 -549.447,E2 -549.447} C_VEL
LIN {X 0,Y 607.782,Z 241.594,A -85,B 0,C 180,E1 -549.999,E2 -549.999} C_VEL
LIN {X 0,Y 604.925,Z 241.949,A -85,B 0,C 180,E1 -550.896,E2 -550.896} C_VEL
LIN {X 0,Y 602.523,Z 242.249,A -85,B 0,C 180,E1 -551.617,E2 -551.617} C_VEL
LIN {X 0,Y 601.492,Z 242.377,A -85,B 0,C 180,E1 -552.174,E2 -552.174} C_VEL
LIN {X 0,Y 601.408,Z 242.386,A -85,B 0,C 180,E1 -552.362,E2 -552.362} C_VEL
LIN {X 0,Y 601.427,Z 242.384,A -85,B 0,C 180,E1 -554.895,E2 -554.895} C_VEL
LIN {X 0,Y 601.423,Z 242.385,A -85,B 0,C 180,E1 -556.985,E2 -556.985} C_VEL
LIN {X 0,Y 601.407,Z 242.386,A -85,B 0,C 180,E1 -559.808,E2 -559.808} C_VEL
LIN {X 0,Y 601.411,Z 242.385,A -85,B 0,C 180,E1 -562.681,E2 -562.681} C_VEL
LIN {X 0,Y 601.405,Z 242.386,A -85,B 0,C 180,E1 -564.877,E2 -564.877} C_VEL
LIN {X 0,Y 601.42,Z 242.384,A -85,B 0,C 180,E1 -567.865,E2 -567.865} C_VEL
LIN {X 0,Y 601.424,Z 242.385,A -85,B 0,C 180,E1 -570.162,E2 -570.162} C_VEL
LIN {X 0,Y 601.427,Z 242.383,A -85,B 0,C 180,E1 -572.715,E2 -572.715} C_VEL
LIN {X 0,Y 601.409,Z 242.386,A -85,B 0,C 180,E1 -575.113,E2 -575.113} C_VEL
LIN {X 0,Y 601.43,Z 242.385,A -85,B 0,C 180,E1 -577.417,E2 -577.417} C_VEL
LIN {X 0,Y 601.404,Z 242.386,A -85,B 0,C 180,E1 -579.993,E2 -579.993} C_VEL
LIN {X 0,Y 601.43,Z 242.383,A -85,B 0,C 180,E1 -582.666,E2 -582.666} C_VEL
LIN {X 0,Y 601.416,Z 242.387,A -85,B 0,C 180,E1 -585.48,E2 -585.48} C_VEL
LIN {X 0,Y 601.422,Z 242.386,A -85,B 0,C 180,E1 -588.404,E2 -588.404} C_VEL
LIN {X 0,Y 601.428,Z 242.383,A -85,B 0,C 180,E1 -590.874,E2 -590.874} C_VEL
LIN {X 0,Y 601.436,Z 242.383,A -85,B 0,C 180,E1 -593.731,E2 -593.731} C_VEL
LIN {X 0,Y 601.43,Z 242.385,A -85,B 0,C 180,E1 -596.686,E2 -596.686} C_VEL
LIN {X 0,Y 601.423,Z 242.384,A -85,B 0,C 180,E1 -599.058,E2 -599.058} C_VEL
LIN {X 0,Y 601.43,Z 242.383,A -85,B 0,C 180,E1 -601.372,E2 -601.372} C_VEL
LIN {X 0,Y 601.4,Z 242.389,A -85,B 0,C 180,E1 -603.635,E2 -603.635} C_VEL
LIN {X 0,Y 601.413,Z 242.387,A -85,B 0,C 180,E1 -606.589,E2 -606.589} C_VEL
LIN {X 0,Y 601.429,Z 242.384,A -85,B 0,C 180,E1 -609.477,E2 -609.477} C_VEL
LIN {X 0,Y 601.398,Z 242.388,A -85,B 0,C 180,E1 -611.607,E2 -611.607} C_VEL
LIN {X 0,Y 601.384,Z 244.683,A -85,B 0,C 180,E1 -613.384,E2 -613.384} C_VEL
LIN {X 0,Y 601.378,Z 248.449,A -85,B 0,C 180,E1 -615.916,E2 -615.916} C_VEL
LIN {X 0,Y 601.365,Z 252.349,A -85,B 0,C 180,E1 -618.54,E2 -618.54} C_VEL
LIN {X 0,Y 601.36,Z 256.61,A -85,B 0,C 180,E1 -621.26,E2 -621.26} C_VEL
LIN {X 0,Y 601.332,Z 260.925,A -85,B 0,C 180,E1 -623.961,E2 -623.961} C_VEL
LIN {X 0,Y 601.317,Z 264.196,A -85,B 0,C 180,E1 -625.978,E2 -625.978} C_VEL
LIN {X 0,Y 601.323,Z 268.602,A -85,B 0,C 180,E1 -628.66,E2 -628.66} C_VEL
LIN {X 0,Y 601.344,Z 273.06,A -85,B 0,C 180,E1 -631.338,E2 -631.338} C_VEL
LIN {X 0,Y 601.288,Z 277.574,A -85,B 0,C 180,E1 -634.021,E2 -634.021} C_VEL
LIN {X 0,Y 601.309,Z 278.709,A -85,B 0,C 180,E1 -634.692,E2 -634.692} C_VEL
LIN {X 0,Y 601.453,Z 290.131,A -85,B 0,C 180,E1 -635.027,E2 -635.027} C_VEL
LIN {X 0,Y 601.422,Z 298.765,A -85,B 0,C 180,E1 -635.363,E2 -635.363} C_VEL
LIN {X 0,Y 601.393,Z 307.185,A -85,B 0,C 180,E1 -635.784,E2 -635.784} C_VEL
LIN {X 0,Y 601.371,Z 314.472,A -85,B 0,C 180,E1 -636.232,E2 -636.232} C_VEL
LIN {X 0,Y 601.416,Z 321.991,A -85,B 0,C 180,E1 -636.794,E2 -636.794} C_VEL
LIN {X 0,Y 601.4,Z 328.556,A -85,B 0,C 180,E1 -637.385,E2 -637.385} C_VEL
LIN {X 0,Y 601.398,Z 334.803,A -85,B 0,C 180,E1 -638.06,E2 -638.06} C_VEL
LIN {X 0,Y 601.381,Z 340.006,A -85,B 0,C 180,E1 -638.737,E2 -638.737} C_VEL
LIN {X 0,Y 601.345,Z 344.348,A -85,B 0,C 180,E1 -639.416,E2 -639.416} C_VEL
LIN {X 0,Y 601.335,Z 347.955,A -85,B 0,C 180,E1 -640.096,E2 -640.096} C_VEL
LIN {X 0,Y 601.331,Z 351.608,A -85,B 0,C 180,E1 -640.978,E2 -640.978} C_VEL
LIN {X 0,Y 601.339,Z 353.243,A -85,B 0,C 180,E1 -641.459,E2 -641.459} C_VEL
LIN {X 0,Y 601.351,Z 354.934,A -85,B 0,C 180,E1 -642.143,E2 -642.143} C_VEL
LIN {X 0,Y 601.32,Z 356.108,A -85,B 0,C 180,E1 -642.829,E2 -642.829} C_VEL
LIN {X 0,Y 601.326,Z 356.999,A -85,B 0,C 180,E1 -644.065,E2 -644.065} C_VEL
LIN {X 0,Y 601.312,Z 356.596,A -85,B 0,C 180,E1 -644.899,E2 -644.899} C_VEL
LIN {X 0,Y 601.32,Z 355.641,A -85,B 0,C 180,E1 -645.593,E2 -645.593} C_VEL
LIN {X 0,Y 601.347,Z 353.325,A -85,B 0,C 180,E1 -646.605,E2 -646.605} C_VEL
LIN {X 0,Y 601.326,Z 349.333,A -85,B 0,C 180,E1 -647.689,E2 -647.689} C_VEL
LIN {X 0,Y 601.363,Z 344.751,A -85,B 0,C 180,E1 -648.603,E2 -648.603} C_VEL
LIN {X 0,Y 601.385,Z 339.299,A -85,B 0,C 180,E1 -649.454,E2 -649.454} C_VEL
LIN {X 0,Y 601.387,Z 332.14,A -85,B 0,C 180,E1 -650.344,E2 -650.344} C_VEL
LIN {X 0,Y 601.431,Z 324.395,A -85,B 0,C 180,E1 -651.096,E2 -651.096} C_VEL
LIN {X 0,Y 601.388,Z 316.914,A -85,B 0,C 180,E1 -651.689,E2 -651.689} C_VEL
LIN {X 0,Y 601.422,Z 308.538,A -85,B 0,C 180,E1 -652.229,E2 -652.229} C_VEL
LIN {X 0,Y 601.477,Z 299.788,A -85,B 0,C 180,E1 -652.679,E2 -652.679} C_VEL
LIN {X 0,Y 601.461,Z 290.695,A -85,B 0,C 180,E1 -653.043,E2 -653.043} C_VEL
LIN {X 0,Y 601.509,Z 281.457,A -85,B 0,C 180,E1 -653.314,E2 -653.314} C_VEL
LIN {X 0,Y 601.328,Z 278.722,A -85,B 0,C 180,E1 -653.39,E2 -653.39} C_VEL
LIN {X 0,Y 601.303,Z 274.572,A -85,B 0,C 180,E1 -655.851,E2 -655.851} C_VEL
LIN {X 0,Y 601.33,Z 269.927,A -85,B 0,C 180,E1 -658.631,E2 -658.631} C_VEL
LIN {X 0,Y 601.318,Z 265.29,A -85,B 0,C 180,E1 -661.443,E2 -661.443} C_VEL
LIN {X 0,Y 601.301,Z 261.262,A -85,B 0,C 180,E1 -663.921,E2 -663.921} C_VEL
LIN {X 0,Y 601.292,Z 256.994,A -85,B 0,C 180,E1 -666.589,E2 -666.589} C_VEL
LIN {X 0,Y 601.286,Z 252.999,A -85,B 0,C 180,E1 -669.135,E2 -669.135} C_VEL
LIN {X 0,Y 601.343,Z 249.08,A -85,B 0,C 180,E1 -671.77,E2 -671.77} C_VEL
LIN {X 0,Y 601.401,Z 244.966,A -85,B 0,C 180,E1 -674.536,E2 -674.536} C_VEL
LIN {X 0,Y 601.381,Z 242.39,A -85,B 0,C 180,E1 -676.43,E2 -676.43} C_VEL
LIN {X 0,Y 601.392,Z 242.385,A -85,B 0,C 180,E1 -679.126,E2 -679.126} C_VEL
LIN {X 0,Y 601.412,Z 242.381,A -85,B 0,C 180,E1 -681.734,E2 -681.734} C_VEL
LIN {X 0,Y 601.398,Z 242.389,A -85,B 0,C 180,E1 -684.248,E2 -684.248} C_VEL
LIN {X 0,Y 601.395,Z 242.383,A -85,B 0,C 180,E1 -686.687,E2 -686.687} C_VEL
LIN {X 0,Y 601.4,Z 242.389,A -85,B 0,C 180,E1 -689.059,E2 -689.059} C_VEL
LIN {X 0,Y 601.429,Z 242.379,A -85,B 0,C 180,E1 -691.375,E2 -691.375} C_VEL
LIN {X 0,Y 601.393,Z 242.388,A -85,B 0,C 180,E1 -693.638,E2 -693.638} C_VEL
LIN {X 0,Y 601.397,Z 242.385,A -85,B 0,C 180,E1 -696.591,E2 -696.591} C_VEL
LIN {X 0,Y 601.423,Z 242.38,A -85,B 0,C 180,E1 -699.48,E2 -699.48} C_VEL
LIN {X 0,Y 601.384,Z 242.384,A -85,B 0,C 180,E1 -702.313,E2 -702.313} C_VEL
LIN {X 0,Y 601.397,Z 242.384,A -85,B 0,C 180,E1 -704.41,E2 -704.41} C_VEL
LIN {X 0,Y 601.411,Z 242.381,A -85,B 0,C 180,E1 -707.173,E2 -707.173} C_VEL
LIN {X 0,Y 601.423,Z 242.382,A -85,B 0,C 180,E1 -709.906,E2 -709.906} C_VEL
LIN {X 0,Y 601.437,Z 242.382,A -85,B 0,C 180,E1 -712.616,E2 -712.616} C_VEL
LIN {X 0,Y 601.403,Z 242.382,A -85,B 0,C 180,E1 -715.309,E2 -715.309} C_VEL
LIN {X 0,Y 601.417,Z 242.381,A -85,B 0,C 180,E1 -717.992,E2 -717.992} C_VEL
LIN {X 0,Y 601.453,Z 242.382,A -85,B 0,C 180,E1 -720.671,E2 -720.671} C_VEL
LIN {X 0,Y 601.404,Z 242.383,A -85,B 0,C 180,E1 -723.351,E2 -723.351} C_VEL
LIN {X 0,Y 601.409,Z 242.381,A -85,B 0,C 180,E1 -726.038,E2 -726.038} C_VEL
LIN {X 0,Y 601.432,Z 242.384,A -85,B 0,C 180,E1 -728.739,E2 -728.739} C_VEL
LIN {X 0,Y 601.4,Z 242.385,A -85,B 0,C 180,E1 -731.46,E2 -731.46} C_VEL
LIN {X 0,Y 601.411,Z 242.381,A -85,B 0,C 180,E1 -734.207,E2 -734.207} C_VEL
LIN {X 0,Y 601.419,Z 242.381,A -85,B 0,C 180,E1 -736.987,E2 -736.987} C_VEL
LIN {X 0,Y 601.391,Z 242.389,A -85,B 0,C 180,E1 -739.811,E2 -739.811} C_VEL
LIN {X 0,Y 601.405,Z 242.386,A -85,B 0,C 180,E1 -742.684,E2 -742.684} C_VEL
LIN {X 0,Y 601.392,Z 242.385,A -85,B 0,C 180,E1 -744.88,E2 -744.88} C_VEL
LIN {X 0,Y 601.384,Z 242.388,A -85,B 0,C 180,E1 -747.87,E2 -747.87} C_VEL
LIN {X 0,Y 601.422,Z 242.38,A -85,B 0,C 180,E1 -750.165,E2 -750.165} C_VEL
LIN {X 0,Y 601.422,Z 242.382,A -85,B 0,C 180,E1 -752.718,E2 -752.718} C_VEL
LIN {X 0,Y 601.374,Z 242.387,A -85,B 0,C 180,E1 -755.111,E2 -755.111} C_VEL
LIN {X 0,Y 601.43,Z 242.382,A -85,B 0,C 180,E1 -757.42,E2 -757.42} C_VEL
LIN {X 0,Y 601.408,Z 242.384,A -85,B 0,C 180,E1 -759.996,E2 -759.996} C_VEL
LIN {X 0,Y 601.398,Z 242.383,A -85,B 0,C 180,E1 -762.672,E2 -762.672} C_VEL
LIN {X 0,Y 601.392,Z 242.385,A -85,B 0,C 180,E1 -765.481,E2 -765.481} C_VEL
LIN {X 0,Y 601.421,Z 242.384,A -85,B 0,C 180,E1 -768.408,E2 -768.408} C_VEL
LIN {X 0,Y 601.403,Z 242.383,A -85,B 0,C 180,E1 -770.874,E2 -770.874} C_VEL
LIN {X 0,Y 601.398,Z 242.384,A -85,B 0,C 180,E1 -773.418,E2 -773.418} C_VEL
LIN {X 0,Y 601.429,Z 242.385,A -85,B 0,C 180,E1 -776.065,E2 -776.065} C_VEL
LIN {X 0,Y 601.462,Z 242.594,A -85,B 0,C 180,E1 -777.18,E2 -777.18} C_VEL
LIN {X 0,Y 601.512,Z 249.836,A -85,B 0,C 180,E1 -779.454,E2 -779.454} C_VEL
LIN {X 0,Y 601.49,Z 258.882,A -85,B 0,C 180,E1 -782.137,E2 -782.137} C_VEL
LIN {X 0,Y 601.473,Z 269.103,A -85,B 0,C 180,E1 -785.126,E2 -785.126} C_VEL
LIN {X 0,Y 601.4,Z 279.322,A -85,B 0,C 180,E1 -788.041,E2 -788.041} C_VEL
LIN {X 0,Y 601.372,Z 289.541,A -85,B 0,C 180,E1 -790.901,E2 -790.901} C_VEL
LIN {X 0,Y 601.361,Z 298.616,A -85,B 0,C 180,E1 -793.399,E2 -793.399} C_VEL
LIN {X 0,Y 601.383,Z 308.936,A -85,B 0,C 180,E1 -796.203,E2 -796.203} C_VEL
LIN {X 0,Y 601.368,Z 319.418,A -85,B 0,C 180,E1 -799.016,E2 -799.016} C_VEL
LIN {X 0,Y 601.341,Z 325.306,A -85,B 0,C 180,E1 -800.584,E2 -800.584} C_VEL
LIN {X 0,Y 601.506,Z 338.507,A -85,B 0,C 180,E1 -800.926,E2 -800.926} C_VEL
LIN {X 0,Y 601.447,Z 347.558,A -85,B 0,C 180,E1 -801.264,E2 -801.264} C_VEL
LIN {X 0,Y 601.424,Z 356.252,A -85,B 0,C 180,E1 -801.686,E2 -801.686} C_VEL
LIN {X 0,Y 601.428,Z 364.557,A -85,B 0,C 180,E1 -802.194,E2 -802.194} C_VEL
LIN {X 0,Y 601.414,Z 372.413,A -85,B 0,C 180,E1 -802.784,E2 -802.784} C_VEL
LIN {X 0,Y 601.411,Z 379.605,A -85,B 0,C 180,E1 -803.444,E2 -803.444} C_VEL
LIN {X 0,Y 601.391,Z 387.198,A -85,B 0,C 180,E1 -804.3,E2 -804.3} C_VEL
LIN {X 0,Y 601.38,Z 393.033,A -85,B 0,C 180,E1 -805.141,E2 -805.141} C_VEL
LIN {X 0,Y 601.345,Z 397.635,A -85,B 0,C 180,E1 -805.98,E2 -805.98} C_VEL
LIN {X 0,Y 601.343,Z 400.625,A -85,B 0,C 180,E1 -806.651,E2 -806.651} C_VEL
LIN {X 0,Y 601.326,Z 402.935,A -85,B 0,C 180,E1 -807.321,E2 -807.321} C_VEL
LIN {X 0,Y 601.343,Z 404.681,A -85,B 0,C 180,E1 -807.992,E2 -807.992} C_VEL
LIN {X 0,Y 601.345,Z 405.936,A -85,B 0,C 180,E1 -808.662,E2 -808.662} C_VEL
LIN {X 0,Y 601.335,Z 406.714,A -85,B 0,C 180,E1 -809.331,E2 -809.331} C_VEL
LIN {X 0,Y 601.332,Z 407,A -85,B 0,C 180,E1 -810.001,E2 -810.001} C_VEL
LIN {X 0,Y 601.335,Z 406.713,A -85,B 0,C 180,E1 -810.671,E2 -810.671} C_VEL
LIN {X 0,Y 601.345,Z 405.933,A -85,B 0,C 180,E1 -811.34,E2 -811.34} C_VEL
LIN {X 0,Y 601.343,Z 404.677,A -85,B 0,C 180,E1 -812.01,E2 -812.01} C_VEL
LIN {X 0,Y 601.342,Z 401.783,A -85,B 0,C 180,E1 -813.016,E2 -813.016} C_VEL
LIN {X 0,Y 601.364,Z 399.143,A -85,B 0,C 180,E1 -813.686,E2 -813.686} C_VEL
LIN {X 0,Y 601.341,Z 393.98,A -85,B 0,C 180,E1 -814.693,E2 -814.693} C_VEL
LIN {X 0,Y 601.383,Z 388.424,A -85,B 0,C 180,E1 -815.533,E2 -815.533} C_VEL
LIN {X 0,Y 601.394,Z 381.156,A -85,B 0,C 180,E1 -816.403,E2 -816.403} C_VEL
LIN {X 0,Y 601.417,Z 373.406,A -85,B 0,C 180,E1 -817.133,E2 -817.133} C_VEL
LIN {X 0,Y 601.413,Z 365.75,A -85,B 0,C 180,E1 -817.724,E2 -817.724} C_VEL
LIN {X 0,Y 601.434,Z 357.708,A -85,B 0,C 180,E1 -818.231,E2 -818.231} C_VEL
LIN {X 0,Y 601.458,Z 349.374,A -85,B 0,C 180,E1 -818.653,E2 -818.653} C_VEL
LIN {X 0,Y 601.469,Z 340.867,A -85,B 0,C 180,E1 -818.992,E2 -818.992} C_VEL
LIN {X 0,Y 601.503,Z 331.553,A -85,B 0,C 180,E1 -819.267,E2 -819.267} C_VEL
LIN {X 0,Y 601.34,Z 325.299,A -85,B 0,C 180,E1 -819.418,E2 -819.418} C_VEL
LIN {X 0,Y 601.367,Z 315.081,A -85,B 0,C 180,E1 -822.144,E2 -822.144} C_VEL
LIN {X 0,Y 601.352,Z 304.862,A -85,B 0,C 180,E1 -824.9,E2 -824.9} C_VEL
LIN {X 0,Y 601.403,Z 294.643,A -85,B 0,C 180,E1 -827.689,E2 -827.689} C_VEL
LIN {X 0,Y 601.389,Z 284.425,A -85,B 0,C 180,E1 -830.524,E2 -830.524} C_VEL
LIN {X 0,Y 601.439,Z 274.206,A -85,B 0,C 180,E1 -833.41,E2 -833.41} C_VEL
LIN {X 0,Y 601.431,Z 265.675,A -85,B 0,C 180,E1 -835.871,E2 -835.871} C_VEL
LIN {X 0,Y 601.501,Z 256.219,A -85,B 0,C 180,E1 -838.624,E2 -838.624} C_VEL
LIN {X 0,Y 601.504,Z 246.899,A -85,B 0,C 180,E1 -841.467,E2 -841.467} C_VEL
LIN {X 0,Y 601.438,Z 242.384,A -85,B 0,C 180,E1 -842.904,E2 -842.904} C_VEL
LIN {X 0,Y 601.389,Z 242.388,A -85,B 0,C 180,E1 -845.755,E2 -845.755} C_VEL
LIN {X 0,Y 601.437,Z 242.383,A -85,B 0,C 180,E1 -848.471,E2 -848.471} C_VEL
LIN {X 0,Y 601.429,Z 242.384,A -85,B 0,C 180,E1 -851.593,E2 -851.593} C_VEL
LIN {X 0,Y 601.404,Z 242.388,A -85,B 0,C 180,E1 -854.533,E2 -854.533} C_VEL
LIN {X 0,Y 601.415,Z 242.387,A -85,B 0,C 180,E1 -857.41,E2 -857.41} C_VEL
LIN {X 0,Y 601.407,Z 242.386,A -85,B 0,C 180,E1 -860.004,E2 -860.004} C_VEL
LIN {X 0,Y 601.44,Z 242.383,A -85,B 0,C 180,E1 -862.618,E2 -862.618} C_VEL
LIN {X 0,Y 601.432,Z 242.383,A -85,B 0,C 180,E1 -865.881,E2 -865.881} C_VEL
LIN {X 0,Y 601.426,Z 242.386,A -85,B 0,C 180,E1 -868.545,E2 -868.545} C_VEL
LIN {X 0,Y 601.433,Z 242.383,A -85,B 0,C 180,E1 -871.373,E2 -871.373} C_VEL
LIN {X 0,Y 601.422,Z 242.384,A -85,B 0,C 180,E1 -874.132,E2 -874.132} C_VEL
LIN {X 0,Y 601.402,Z 242.388,A -85,B 0,C 180,E1 -876.588,E2 -876.588} C_VEL
LIN {X 0,Y 601.431,Z 242.384,A -85,B 0,C 180,E1 -879.477,E2 -879.477} C_VEL
LIN {X 0,Y 601.405,Z 242.386,A -85,B 0,C 180,E1 -882.311,E2 -882.311} C_VEL
LIN {X 0,Y 601.419,Z 242.384,A -85,B 0,C 180,E1 -884.408,E2 -884.408} C_VEL
LIN {X 0,Y 601.421,Z 242.384,A -85,B 0,C 180,E1 -887.171,E2 -887.171} C_VEL
LIN {X 0,Y 601.428,Z 242.385,A -85,B 0,C 180,E1 -889.904,E2 -889.904} C_VEL
LIN {X 0,Y 601.444,Z 242.382,A -85,B 0,C 180,E1 -892.614,E2 -892.614} C_VEL
LIN {X 0,Y 601.426,Z 242.383,A -85,B 0,C 180,E1 -895.307,E2 -895.307} C_VEL
LIN {X 0,Y 601.429,Z 242.385,A -85,B 0,C 180,E1 -897.99,E2 -897.99} C_VEL
LIN {X 0,Y 601.449,Z 242.381,A -85,B 0,C 180,E1 -900.668,E2 -900.668} C_VEL
LIN {X 0,Y 601.438,Z 242.382,A -85,B 0,C 180,E1 -903.348,E2 -903.348} C_VEL
LIN {X 0,Y 601.417,Z 242.387,A -85,B 0,C 180,E1 -906.036,E2 -906.036} C_VEL
LIN {X 0,Y 601.413,Z 242.385,A -85,B 0,C 180,E1 -908.737,E2 -908.737} C_VEL
LIN {X 0,Y 601.44,Z 242.382,A -85,B 0,C 180,E1 -911.457,E2 -911.457} C_VEL
LIN {X 0,Y 601.408,Z 242.386,A -85,B 0,C 180,E1 -912.362,E2 -912.362} C_VEL
LIN {X 0,Y 600.741,Z 242.47,A -85,B 0,C 180,E1 -912.922,E2 -912.922} C_VEL
LIN {X 0,Y 597.892,Z 242.825,A -85,B 0,C 180,E1 -913.83,E2 -913.83} C_VEL
LIN {X 0,Y 595.483,Z 243.126,A -85,B 0,C 180,E1 -914.56,E2 -914.56} C_VEL
LIN {X 0,Y 594.447,Z 243.255,A -85,B 0,C 180,E1 -915.124,E2 -915.124} C_VEL
LIN {X 0,Y 594.361,Z 243.264,A -85,B 0,C 180,E1 -915.314,E2 -915.314} C_VEL
LIN {X 0,Y 594.385,Z 243.262,A -85,B 0,C 180,E1 -917.192,E2 -917.192} C_VEL
LIN {X 0,Y 594.376,Z 243.263,A -85,B 0,C 180,E1 -920.052,E2 -920.052} C_VEL
LIN {X 0,Y 594.364,Z 243.264,A -85,B 0,C 180,E1 -922.965,E2 -922.965} C_VEL
LIN {X 0,Y 594.375,Z 243.264,A -85,B 0,C 180,E1 -925.191,E2 -925.191} C_VEL
LIN {X 0,Y 594.383,Z 243.261,A -85,B 0,C 180,E1 -927.525,E2 -927.525} C_VEL
LIN {X 0,Y 594.384,Z 243.262,A -85,B 0,C 180,E1 -930.327,E2 -930.327} C_VEL
LIN {X 0,Y 594.377,Z 243.261,A -85,B 0,C 180,E1 -932.948,E2 -932.948} C_VEL
LIN {X 0,Y 594.377,Z 243.263,A -85,B 0,C 180,E1 -935.405,E2 -935.405} C_VEL
LIN {X 0,Y 594.381,Z 243.261,A -85,B 0,C 180,E1 -937.939,E2 -937.939} C_VEL
LIN {X 0,Y 594.374,Z 243.262,A -85,B 0,C 180,E1 -940.821,E2 -940.821} C_VEL
LIN {X 0,Y 594.378,Z 243.263,A -85,B 0,C 180,E1 -943.296,E2 -943.296} C_VEL
LIN {X 0,Y 594.372,Z 243.262,A -85,B 0,C 180,E1 -946.157,E2 -946.157} C_VEL
LIN {X 0,Y 594.379,Z 243.263,A -85,B 0,C 180,E1 -948.535,E2 -948.535} C_VEL
LIN {X 0,Y 594.38,Z 243.262,A -85,B 0,C 180,E1 -951.293,E2 -951.293} C_VEL
LIN {X 0,Y 594.388,Z 243.261,A -85,B 0,C 180,E1 -953.757,E2 -953.757} C_VEL
LIN {X 0,Y 594.38,Z 243.261,A -85,B 0,C 180,E1 -956.238,E2 -956.238} C_VEL
LIN {X 0,Y 594.382,Z 243.263,A -85,B 0,C 180,E1 -958.65,E2 -958.65} C_VEL
LIN {X 0,Y 594.378,Z 243.261,A -85,B 0,C 180,E1 -961.038,E2 -961.038} C_VEL
LIN {X 0,Y 594.382,Z 243.261,A -85,B 0,C 180,E1 -963.973,E2 -963.973} C_VEL
LIN {X 0,Y 594.383,Z 243.261,A -85,B 0,C 180,E1 -966.295,E2 -966.295} C_VEL
LIN {X 0,Y 594.399,Z 243.258,A -85,B 0,C 180,E1 -969.224,E2 -969.224} C_VEL
LIN {X 0,Y 594.373,Z 243.262,A -85,B 0,C 180,E1 -971.381,E2 -971.381} C_VEL
LIN {X 0,Y 594.305,Z 243.454,A -85,B 0,C 180,E1 -972.093,E2 -972.093} C_VEL
LIN {X 0,Y 594.29,Z 246.56,A -85,B 0,C 180,E1 -974.216,E2 -974.216} C_VEL
LIN {X 0,Y 594.287,Z 249.653,A -85,B 0,C 180,E1 -976.318,E2 -976.318} C_VEL
LIN {X 0,Y 594.292,Z 253.704,A -85,B 0,C 180,E1 -979.092,E2 -979.092} C_VEL
LIN {X 0,Y 594.271,Z 257.967,A -85,B 0,C 180,E1 -981.841,E2 -981.841} C_VEL
LIN {X 0,Y 594.257,Z 261.207,A -85,B 0,C 180,E1 -983.889,E2 -983.889} C_VEL
LIN {X 0,Y 594.235,Z 264.478,A -85,B 0,C 180,E1 -985.93,E2 -985.93} C_VEL
LIN {X 0,Y 594.23,Z 268.884,A -85,B 0,C 180,E1 -988.644,E2 -988.644} C_VEL
LIN {X 0,Y 594.246,Z 273.342,A -85,B 0,C 180,E1 -991.354,E2 -991.354} C_VEL
LIN {X 0,Y 594.204,Z 277.855,A -85,B 0,C 180,E1 -994.069,E2 -994.069} C_VEL
LIN {X 0,Y 594.228,Z 278.706,A -85,B 0,C 180,E1 -994.578,E2 -994.578} C_VEL
LIN {X 0,Y 594.504,Z 285.388,A -85,B 0,C 180,E1 -994.767,E2 -994.767} C_VEL
LIN {X 0,Y 594.43,Z 296.83,A -85,B 0,C 180,E1 -995.171,E2 -995.171} C_VEL
LIN {X 0,Y 594.363,Z 307.133,A -85,B 0,C 180,E1 -995.682,E2 -995.682} C_VEL
LIN {X 0,Y 594.321,Z 315.394,A -85,B 0,C 180,E1 -996.203,E2 -996.203} C_VEL
LIN {X 0,Y 594.366,Z 322.968,A -85,B 0,C 180,E1 -996.79,E2 -996.79} C_VEL
LIN {X 0,Y 594.327,Z 330.229,A -85,B 0,C 180,E1 -997.473,E2 -997.473} C_VEL
LIN {X 0,Y 594.282,Z 337.597,A -85,B 0,C 180,E1 -998.329,E2 -998.329} C_VEL
LIN {X 0,Y 594.275,Z 343.362,A -85,B 0,C 180,E1 -999.186,E2 -999.186} C_VEL
LIN {X 0,Y 594.253,Z 347.166,A -85,B 0,C 180,E1 -999.873,E2 -999.873} C_VEL
LIN {X 0,Y 594.233,Z 351.493,A -85,B 0,C 180,E1 -1000.907,E2 -1000.907} C_VEL
LIN {X 0,Y 594.262,Z 353.699,A -85,B 0,C 180,E1 -1001.597,E2 -1001.597} C_VEL
LIN {X 0,Y 594.242,Z 355.327,A -85,B 0,C 180,E1 -1002.29,E2 -1002.29} C_VEL
LIN {X 0,Y 594.236,Z 356.344,A -85,B 0,C 180,E1 -1002.985,E2 -1002.985} C_VEL
LIN {X 0,Y 594.237,Z 356.986,A -85,B 0,C 180,E1 -1004.125,E2 -1004.125} C_VEL
LIN {X 0,Y 594.222,Z 356.378,A -85,B 0,C 180,E1 -1005.081,E2 -1005.081} C_VEL
LIN {X 0,Y 594.249,Z 355.36,A -85,B 0,C 180,E1 -1005.783,E2 -1005.783} C_VEL
LIN {X 0,Y 594.255,Z 353.179,A -85,B 0,C 180,E1 -1006.683,E2 -1006.683} C_VEL
LIN {X 0,Y 594.254,Z 350.143,A -85,B 0,C 180,E1 -1007.551,E2 -1007.551} C_VEL
LIN {X 0,Y 594.265,Z 346.94,A -85,B 0,C 180,E1 -1008.263,E2 -1008.263} C_VEL
LIN {X 0,Y 594.31,Z 342.289,A -85,B 0,C 180,E1 -1009.084,E2 -1009.084} C_VEL
LIN {X 0,Y 594.305,Z 336.692,A -85,B 0,C 180,E1 -1009.875,E2 -1009.875} C_VEL
LIN {X 0,Y 594.325,Z 330.436,A -85,B 0,C 180,E1 -1010.596,E2 -1010.596} C_VEL
LIN {X 0,Y 594.386,Z 324.525,A -85,B 0,C 180,E1 -1011.169,E2 -1011.169} C_VEL
LIN {X 0,Y 594.342,Z 316.963,A -85,B 0,C 180,E1 -1011.776,E2 -1011.776} C_VEL
LIN {X 0,Y 594.4,Z 308.899,A -85,B 0,C 180,E1 -1012.305,E2 -1012.305} C_VEL
LIN {X 0,Y 594.461,Z 300.201,A -85,B 0,C 180,E1 -1012.763,E2 -1012.763} C_VEL
LIN {X 0,Y 594.45,Z 292.088,A -85,B 0,C 180,E1 -1013.101,E2 -1013.101} C_VEL
LIN {X 0,Y 594.504,Z 283.381,A -85,B 0,C 180,E1 -1013.375,E2 -1013.375} C_VEL
LIN {X 0,Y 594.223,Z 278.723,A -85,B 0,C 180,E1 -1013.502,E2 -1013.502} C_VEL
LIN {X 0,Y 594.201,Z 274.577,A -85,B 0,C 180,E1 -1015.991,E2 -1015.991} C_VEL
LIN {X 0,Y 594.214,Z 270.872,A -85,B 0,C 180,E1 -1018.234,E2 -1018.234} C_VEL
LIN {X 0,Y 594.231,Z 267.057,A -85,B 0,C 180,E1 -1020.567,E2 -1020.567} C_VEL
LIN {X 0,Y 594.237,Z 263.195,A -85,B 0,C 180,E1 -1022.958,E2 -1022.958} C_VEL
LIN {X 0,Y 594.202,Z 259.281,A -85,B 0,C 180,E1 -1025.418,E2 -1025.418} C_VEL
LIN {X 0,Y 594.238,Z 255.316,A -85,B 0,C 180,E1 -1027.95,E2 -1027.95} C_VEL
LIN {X 0,Y 594.247,Z 251.15,A -85,B 0,C 180,E1 -1030.811,E2 -1030.811} C_VEL
LIN {X 0,Y 594.309,Z 247.44,A -85,B 0,C 180,E1 -1033.303,E2 -1033.303} C_VEL
LIN {X 0,Y 594.311,Z 243.272,A -85,B 0,C 180,E1 -1036.164,E2 -1036.164} C_VEL
LIN {X 0,Y 594.357,Z 243.26,A -85,B 0,C 180,E1 -1038.537,E2 -1038.537} C_VEL
LIN {X 0,Y 594.374,Z 243.262,A -85,B 0,C 180,E1 -1041.295,E2 -1041.295} C_VEL
LIN {X 0,Y 594.383,Z 243.257,A -85,B 0,C 180,E1 -1043.76,E2 -1043.76} C_VEL
LIN {X 0,Y 594.357,Z 243.262,A -85,B 0,C 180,E1 -1046.24,E2 -1046.24} C_VEL
LIN {X 0,Y 594.351,Z 243.262,A -85,B 0,C 180,E1 -1048.651,E2 -1048.651} C_VEL
LIN {X 0,Y 594.376,Z 243.259,A -85,B 0,C 180,E1 -1051.041,E2 -1051.041} C_VEL
LIN {X 0,Y 594.366,Z 243.262,A -85,B 0,C 180,E1 -1053.978,E2 -1053.978} C_VEL
LIN {X 0,Y 594.363,Z 243.259,A -85,B 0,C 180,E1 -1056.297,E2 -1056.297} C_VEL
LIN {X 0,Y 594.395,Z 243.255,A -85,B 0,C 180,E1 -1059.226,E2 -1059.226} C_VEL
LIN {X 0,Y 594.367,Z 243.26,A -85,B 0,C 180,E1 -1062.097,E2 -1062.097} C_VEL
LIN {X 0,Y 594.348,Z 243.261,A -85,B 0,C 180,E1 -1064.22,E2 -1064.22} C_VEL
LIN {X 0,Y 594.359,Z 243.26,A -85,B 0,C 180,E1 -1067.018,E2 -1067.018} C_VEL
LIN {X 0,Y 594.385,Z 243.26,A -85,B 0,C 180,E1 -1069.785,E2 -1069.785} C_VEL
LIN {X 0,Y 594.383,Z 243.26,A -85,B 0,C 180,E1 -1072.528,E2 -1072.528} C_VEL
LIN {X 0,Y 594.374,Z 243.258,A -85,B 0,C 180,E1 -1075.254,E2 -1075.254} C_VEL
LIN {X 0,Y 594.387,Z 243.257,A -85,B 0,C 180,E1 -1077.968,E2 -1077.968} C_VEL
LIN {X 0,Y 594.421,Z 243.258,A -85,B 0,C 180,E1 -1080.679,E2 -1080.679} C_VEL
LIN {X 0,Y 594.357,Z 243.261,A -85,B 0,C 180,E1 -1083.391,E2 -1083.391} C_VEL
LIN {X 0,Y 594.365,Z 243.259,A -85,B 0,C 180,E1 -1086.11,E2 -1086.11} C_VEL
LIN {X 0,Y 594.388,Z 243.259,A -85,B 0,C 180,E1 -1088.843,E2 -1088.843} C_VEL
LIN {X 0,Y 594.37,Z 243.262,A -85,B 0,C 180,E1 -1091.597,E2 -1091.597} C_VEL
LIN {X 0,Y 594.381,Z 243.257,A -85,B 0,C 180,E1 -1094.378,E2 -1094.378} C_VEL
LIN {X 0,Y 594.376,Z 243.257,A -85,B 0,C 180,E1 -1097.195,E2 -1097.195} C_VEL
LIN {X 0,Y 594.36,Z 243.262,A -85,B 0,C 180,E1 -1100.055,E2 -1100.055} C_VEL
LIN {X 0,Y 594.359,Z 243.265,A -85,B 0,C 180,E1 -1102.968,E2 -1102.968} C_VEL
LIN {X 0,Y 594.368,Z 243.258,A -85,B 0,C 180,E1 -1105.194,E2 -1105.194} C_VEL
LIN {X 0,Y 594.341,Z 243.267,A -85,B 0,C 180,E1 -1107.521,E2 -1107.521} C_VEL
LIN {X 0,Y 594.381,Z 243.258,A -85,B 0,C 180,E1 -1110.33,E2 -1110.33} C_VEL
LIN {X 0,Y 594.375,Z 243.258,A -85,B 0,C 180,E1 -1112.951,E2 -1112.951} C_VEL
LIN {X 0,Y 594.337,Z 243.267,A -85,B 0,C 180,E1 -1115.411,E2 -1115.411} C_VEL
LIN {X 0,Y 594.376,Z 243.257,A -85,B 0,C 180,E1 -1117.942,E2 -1117.942} C_VEL
LIN {X 0,Y 594.375,Z 243.258,A -85,B 0,C 180,E1 -1120.824,E2 -1120.824} C_VEL
LIN {X 0,Y 594.353,Z 243.263,A -85,B 0,C 180,E1 -1123.84,E2 -1123.84} C_VEL
LIN {X 0,Y 594.362,Z 243.266,A -85,B 0,C 180,E1 -1126.702,E2 -1126.702} C_VEL
LIN {X 0,Y 594.386,Z 243.258,A -85,B 0,C 180,E1 -1129.436,E2 -1129.436} C_VEL
LIN {X 0,Y 594.378,Z 243.258,A -85,B 0,C 180,E1 -1132.393,E2 -1132.393} C_VEL
LIN {X 0,Y 594.377,Z 243.258,A -85,B 0,C 180,E1 -1135.421,E2 -1135.421} C_VEL
LIN {X 0,Y 594.394,Z 243.263,A -85,B 0,C 180,E1 -1136.951,E2 -1136.951} C_VEL
LIN {X 0,Y 594.547,Z 249.833,A -85,B 0,C 180,E1 -1139.057,E2 -1139.057} C_VEL
LIN {X 0,Y 594.476,Z 258.763,A -85,B 0,C 180,E1 -1141.779,E2 -1141.779} C_VEL
LIN {X 0,Y 594.447,Z 267.826,A -85,B 0,C 180,E1 -1144.437,E2 -1144.437} C_VEL
LIN {X 0,Y 594.367,Z 277.569,A -85,B 0,C 180,E1 -1147.265,E2 -1147.265} C_VEL
LIN {X 0,Y 594.356,Z 286.986,A -85,B 0,C 180,E1 -1149.947,E2 -1149.947} C_VEL
LIN {X 0,Y 594.309,Z 297.205,A -85,B 0,C 180,E1 -1152.805,E2 -1152.805} C_VEL
LIN {X 0,Y 594.311,Z 307.423,A -85,B 0,C 180,E1 -1155.622,E2 -1155.622} C_VEL
LIN {X 0,Y 594.298,Z 317.642,A -85,B 0,C 180,E1 -1158.403,E2 -1158.403} C_VEL
LIN {X 0,Y 594.268,Z 325.306,A -85,B 0,C 180,E1 -1160.471,E2 -1160.471} C_VEL
LIN {X 0,Y 594.489,Z 338.505,A -85,B 0,C 180,E1 -1160.818,E2 -1160.818} C_VEL
LIN {X 0,Y 594.44,Z 347.555,A -85,B 0,C 180,E1 -1161.16,E2 -1161.16} C_VEL
LIN {X 0,Y 594.399,Z 356.254,A -85,B 0,C 180,E1 -1161.587,E2 -1161.587} C_VEL
LIN {X 0,Y 594.393,Z 364.559,A -85,B 0,C 180,E1 -1162.101,E2 -1162.101} C_VEL
LIN {X 0,Y 594.355,Z 372.413,A -85,B 0,C 180,E1 -1162.698,E2 -1162.698} C_VEL
LIN {X 0,Y 594.342,Z 379.523,A -85,B 0,C 180,E1 -1163.357,E2 -1163.357} C_VEL
LIN {X 0,Y 594.318,Z 387.198,A -85,B 0,C 180,E1 -1164.232,E2 -1164.232} C_VEL
LIN {X 0,Y 594.289,Z 393.033,A -85,B 0,C 180,E1 -1165.082,E2 -1165.082} C_VEL
LIN {X 0,Y 594.261,Z 397.635,A -85,B 0,C 180,E1 -1165.932,E2 -1165.932} C_VEL
LIN {X 0,Y 594.265,Z 400.625,A -85,B 0,C 180,E1 -1166.611,E2 -1166.611} C_VEL
LIN {X 0,Y 594.228,Z 402.935,A -85,B 0,C 180,E1 -1167.289,E2 -1167.289} C_VEL
LIN {X 0,Y 594.242,Z 404.682,A -85,B 0,C 180,E1 -1167.968,E2 -1167.968} C_VEL
LIN {X 0,Y 594.245,Z 405.936,A -85,B 0,C 180,E1 -1168.646,E2 -1168.646} C_VEL
LIN {X 0,Y 594.235,Z 406.713,A -85,B 0,C 180,E1 -1169.323,E2 -1169.323} C_VEL
LIN {X 0,Y 594.233,Z 407,A -85,B 0,C 180,E1 -1170.001,E2 -1170.001} C_VEL
LIN {X 0,Y 594.235,Z 406.712,A -85,B 0,C 180,E1 -1170.679,E2 -1170.679} C_VEL
LIN {X 0,Y 594.245,Z 405.934,A -85,B 0,C 180,E1 -1171.356,E2 -1171.356} C_VEL
LIN {X 0,Y 594.242,Z 404.677,A -85,B 0,C 180,E1 -1172.034,E2 -1172.034} C_VEL
LIN {X 0,Y 594.245,Z 401.784,A -85,B 0,C 180,E1 -1173.052,E2 -1173.052} C_VEL
LIN {X 0,Y 594.286,Z 399.143,A -85,B 0,C 180,E1 -1173.73,E2 -1173.73} C_VEL
LIN {X 0,Y 594.256,Z 393.98,A -85,B 0,C 180,E1 -1174.75,E2 -1174.75} C_VEL
LIN {X 0,Y 594.319,Z 387.182,A -85,B 0,C 180,E1 -1175.77,E2 -1175.77} C_VEL
LIN {X 0,Y 594.343,Z 379.511,A -85,B 0,C 180,E1 -1176.644,E2 -1176.644} C_VEL
LIN {X 0,Y 594.356,Z 372.394,A -85,B 0,C 180,E1 -1177.304,E2 -1177.304} C_VEL
LIN {X 0,Y 594.394,Z 364.535,A -85,B 0,C 180,E1 -1177.901,E2 -1177.901} C_VEL
LIN {X 0,Y 594.42,Z 354.723,A -85,B 0,C 180,E1 -1178.5,E2 -1178.5} C_VEL
LIN {X 0,Y 594.465,Z 343.274,A -85,B 0,C 180,E1 -1179.013,E2 -1179.013} C_VEL
LIN {X 0,Y 594.492,Z 333.214,A -85,B 0,C 180,E1 -1179.334,E2 -1179.334} C_VEL
LIN {X 0,Y 594.268,Z 325.299,A -85,B 0,C 180,E1 -1179.531,E2 -1179.531} C_VEL
LIN {X 0,Y 594.301,Z 315.081,A -85,B 0,C 180,E1 -1182.291,E2 -1182.291} C_VEL
LIN {X 0,Y 594.291,Z 304.862,A -85,B 0,C 180,E1 -1185.081,E2 -1185.081} C_VEL
LIN {X 0,Y 594.35,Z 294.643,A -85,B 0,C 180,E1 -1187.906,E2 -1187.906} C_VEL
LIN {X 0,Y 594.344,Z 285.702,A -85,B 0,C 180,E1 -1190.417,E2 -1190.417} C_VEL
LIN {X 0,Y 594.421,Z 275.483,A -85,B 0,C 180,E1 -1193.334,E2 -1193.334} C_VEL
LIN {X 0,Y 594.458,Z 265.202,A -85,B 0,C 180,E1 -1196.323,E2 -1196.323} C_VEL
LIN {X 0,Y 594.512,Z 256.187,A -85,B 0,C 180,E1 -1198.992,E2 -1198.992} C_VEL
LIN {X 0,Y 594.534,Z 247.563,A -85,B 0,C 180,E1 -1201.667,E2 -1201.667} C_VEL
LIN {X 0,Y 594.397,Z 243.261,A -85,B 0,C 180,E1 -1203.051,E2 -1203.051} C_VEL
LIN {X 0,Y 594.354,Z 243.266,A -85,B 0,C 180,E1 -1205.409,E2 -1205.409} C_VEL
LIN {X 0,Y 594.39,Z 243.26,A -85,B 0,C 180,E1 -1207.941,E2 -1207.941} C_VEL
LIN {X 0,Y 594.383,Z 243.26,A -85,B 0,C 180,E1 -1210.822,E2 -1210.822} C_VEL
LIN {X 0,Y 594.373,Z 243.263,A -85,B 0,C 180,E1 -1213.3,E2 -1213.3} C_VEL
LIN {X 0,Y 594.367,Z 243.263,A -85,B 0,C 180,E1 -1216.161,E2 -1216.161} C_VEL
LIN {X 0,Y 594.385,Z 243.262,A -85,B 0,C 180,E1 -1218.536,E2 -1218.536} C_VEL
LIN {X 0,Y 594.376,Z 243.262,A -85,B 0,C 180,E1 -1221.297,E2 -1221.297} C_VEL
LIN {X 0,Y 594.355,Z 243.265,A -85,B 0,C 180,E1 -1223.755,E2 -1223.755} C_VEL
LIN {X 0,Y 594.385,Z 243.261,A -85,B 0,C 180,E1 -1226.239,E2 -1226.239} C_VEL
LIN {X 0,Y 594.375,Z 243.264,A -85,B 0,C 180,E1 -1228.649,E2 -1228.649} C_VEL
LIN {X 0,Y 594.387,Z 243.26,A -85,B 0,C 180,E1 -1231.043,E2 -1231.043} C_VEL
LIN {X 0,Y 594.396,Z 243.259,A -85,B 0,C 180,E1 -1233.976,E2 -1233.976} C_VEL
LIN {X 0,Y 594.383,Z 243.26,A -85,B 0,C 180,E1 -1236.295,E2 -1236.295} C_VEL
LIN {X 0,Y 594.404,Z 243.258,A -85,B 0,C 180,E1 -1239.224,E2 -1239.224} C_VEL
LIN {X 0,Y 594.36,Z 243.263,A -85,B 0,C 180,E1 -1242.094,E2 -1242.094} C_VEL
LIN {X 0,Y 594.372,Z 243.262,A -85,B 0,C 180,E1 -1244.218,E2 -1244.218} C_VEL
LIN {X 0,Y 594.369,Z 243.263,A -85,B 0,C 180,E1 -1247.016,E2 -1247.016} C_VEL
LIN {X 0,Y 594.389,Z 243.262,A -85,B 0,C 180,E1 -1249.783,E2 -1249.783} C_VEL
LIN {X 0,Y 594.398,Z 243.259,A -85,B 0,C 180,E1 -1252.526,E2 -1252.526} C_VEL
LIN {X 0,Y 594.396,Z 243.259,A -85,B 0,C 180,E1 -1255.251,E2 -1255.251} C_VEL
LIN {X 0,Y 594.4,Z 243.261,A -85,B 0,C 180,E1 -1257.966,E2 -1257.966} C_VEL
LIN {X 0,Y 594.421,Z 243.257,A -85,B 0,C 180,E1 -1260.676,E2 -1260.676} C_VEL
LIN {X 0,Y 594.389,Z 243.26,A -85,B 0,C 180,E1 -1263.388,E2 -1263.388} C_VEL
LIN {X 0,Y 594.371,Z 243.264,A -85,B 0,C 180,E1 -1266.108,E2 -1266.108} C_VEL
LIN {X 0,Y 594.382,Z 243.262,A -85,B 0,C 180,E1 -1268.841,E2 -1268.841} C_VEL
LIN {X 0,Y 594.398,Z 243.259,A -85,B 0,C 180,E1 -1271.594,E2 -1271.594} C_VEL
LIN {X 0,Y 594.39,Z 243.26,A -85,B 0,C 180,E1 -1274.375,E2 -1274.375} C_VEL
LIN {X 0,Y 594.361,Z 243.264,A -85,B 0,C 180,E1 -1275.314,E2 -1275.314} C_VEL
LIN {X 0,Y 593.688,Z 243.349,A -85,B 0,C 180,E1 -1275.88,E2 -1275.88} C_VEL
LIN {X 0,Y 590.822,Z 243.706,A -85,B 0,C 180,E1 -1276.798,E2 -1276.798} C_VEL
LIN {X 0,Y 588.412,Z 244.008,A -85,B 0,C 180,E1 -1277.537,E2 -1277.537} C_VEL
LIN {X 0,Y 587.388,Z 244.134,A -85,B 0,C 180,E1 -1278.107,E2 -1278.107} C_VEL
LIN {X 0,Y 587.311,Z 244.143,A -85,B 0,C 180,E1 -1278.3,E2 -1278.3} C_VEL
LIN {X 0,Y 587.33,Z 244.141,A -85,B 0,C 180,E1 -1281.036,E2 -1281.036} C_VEL
LIN {X 0,Y 587.322,Z 244.142,A -85,B 0,C 180,E1 -1283.257,E2 -1283.257} C_VEL
LIN {X 0,Y 587.332,Z 244.139,A -85,B 0,C 180,E1 -1285.515,E2 -1285.515} C_VEL
LIN {X 0,Y 587.347,Z 244.137,A -85,B 0,C 180,E1 -1287.816,E2 -1287.816} C_VEL
LIN {X 0,Y 587.34,Z 244.138,A -85,B 0,C 180,E1 -1290.509,E2 -1290.509} C_VEL
LIN {X 0,Y 587.337,Z 244.139,A -85,B 0,C 180,E1 -1293.11,E2 -1293.11} C_VEL
LIN {X 0,Y 587.351,Z 244.137,A -85,B 0,C 180,E1 -1295.893,E2 -1295.893} C_VEL
LIN {X 0,Y 587.326,Z 244.141,A -85,B 0,C 180,E1 -1298.477,E2 -1298.477} C_VEL
LIN {X 0,Y 587.331,Z 244.14,A -85,B 0,C 180,E1 -1301.155,E2 -1301.155} C_VEL
LIN {X 0,Y 587.325,Z 244.14,A -85,B 0,C 180,E1 -1304.112,E2 -1304.112} C_VEL
LIN {X 0,Y 587.326,Z 244.14,A -85,B 0,C 180,E1 -1306.994,E2 -1306.994} C_VEL
LIN {X 0,Y 587.32,Z 244.141,A -85,B 0,C 180,E1 -1309.745,E2 -1309.745} C_VEL
LIN {X 0,Y 587.337,Z 244.139,A -85,B 0,C 180,E1 -1312.391,E2 -1312.391} C_VEL
LIN {X 0,Y 587.34,Z 244.138,A -85,B 0,C 180,E1 -1314.945,E2 -1314.945} C_VEL
LIN {X 0,Y 587.336,Z 244.14,A -85,B 0,C 180,E1 -1317.42,E2 -1317.42} C_VEL
LIN {X 0,Y 587.335,Z 244.139,A -85,B 0,C 180,E1 -1319.829,E2 -1319.829} C_VEL
LIN {X 0,Y 587.337,Z 244.138,A -85,B 0,C 180,E1 -1322.305,E2 -1322.305} C_VEL
LIN {X 0,Y 587.328,Z 244.14,A -85,B 0,C 180,E1 -1324.482,E2 -1324.482} C_VEL
LIN {X 0,Y 587.357,Z 244.137,A -85,B 0,C 180,E1 -1327.486,E2 -1327.486} C_VEL
LIN {X 0,Y 587.335,Z 244.139,A -85,B 0,C 180,E1 -1330.424,E2 -1330.424} C_VEL
LIN {X 0,Y 587.257,Z 244.15,A -85,B 0,C 180,E1 -1331.87,E2 -1331.87} C_VEL
LIN {X 0,Y 587.276,Z 245.882,A -85,B 0,C 180,E1 -1333.308,E2 -1333.308} C_VEL
LIN {X 0,Y 587.22,Z 250.017,A -85,B 0,C 180,E1 -1336.15,E2 -1336.15} C_VEL
LIN {X 0,Y 587.248,Z 254.119,A -85,B 0,C 180,E1 -1338.96,E2 -1338.96} C_VEL
LIN {X 0,Y 587.205,Z 258.25,A -85,B 0,C 180,E1 -1341.742,E2 -1341.742} C_VEL
LIN {X 0,Y 587.188,Z 261.489,A -85,B 0,C 180,E1 -1343.815,E2 -1343.815} C_VEL
LIN {X 0,Y 587.157,Z 264.759,A -85,B 0,C 180,E1 -1345.881,E2 -1345.881} C_VEL
LIN {X 0,Y 587.136,Z 269.165,A -85,B 0,C 180,E1 -1348.627,E2 -1348.627} C_VEL
LIN {X 0,Y 587.148,Z 273.624,A -85,B 0,C 180,E1 -1351.371,E2 -1351.371} C_VEL
LIN {X 0,Y 587.125,Z 278.137,A -85,B 0,C 180,E1 -1354.118,E2 -1354.118} C_VEL
LIN {X 0,Y 587.142,Z 278.704,A -85,B 0,C 180,E1 -1354.461,E2 -1354.461} C_VEL
LIN {X 0,Y 587.494,Z 284.443,A -85,B 0,C 180,E1 -1354.631,E2 -1354.631} C_VEL
LIN {X 0,Y 587.402,Z 295.807,A -85,B 0,C 180,E1 -1355.018,E2 -1355.018} C_VEL
LIN {X 0,Y 587.339,Z 305.589,A -85,B 0,C 180,E1 -1355.492,E2 -1355.492} C_VEL
LIN {X 0,Y 587.27,Z 314.003,A -85,B 0,C 180,E1 -1356.01,E2 -1356.01} C_VEL
LIN {X 0,Y 587.301,Z 321.44,A -85,B 0,C 180,E1 -1356.572,E2 -1356.572} C_VEL
LIN {X 0,Y 587.274,Z 328.495,A -85,B 0,C 180,E1 -1357.218,E2 -1357.218} C_VEL
LIN {X 0,Y 587.26,Z 334.752,A -85,B 0,C 180,E1 -1357.91,E2 -1357.91} C_VEL
LIN {X 0,Y 587.24,Z 339.961,A -85,B 0,C 180,E1 -1358.603,E2 -1358.603} C_VEL
LIN {X 0,Y 587.194,Z 344.311,A -85,B 0,C 180,E1 -1359.298,E2 -1359.298} C_VEL
LIN {X 0,Y 587.164,Z 349.463,A -85,B 0,C 180,E1 -1360.342,E2 -1360.342} C_VEL
LIN {X 0,Y 587.172,Z 352.121,A -85,B 0,C 180,E1 -1361.057,E2 -1361.057} C_VEL
LIN {X 0,Y 587.17,Z 354.102,A -85,B 0,C 180,E1 -1361.739,E2 -1361.739} C_VEL
LIN {X 0,Y 587.158,Z 355.611,A -85,B 0,C 180,E1 -1362.441,E2 -1362.441} C_VEL
LIN {X 0,Y 587.134,Z 356.57,A -85,B 0,C 180,E1 -1363.145,E2 -1363.145} C_VEL
LIN {X 0,Y 587.136,Z 356.963,A -85,B 0,C 180,E1 -1364.181,E2 -1364.181} C_VEL
LIN {X 0,Y 587.136,Z 356.141,A -85,B 0,C 180,E1 -1365.267,E2 -1365.267} C_VEL
LIN {X 0,Y 587.158,Z 354.969,A -85,B 0,C 180,E1 -1365.979,E2 -1365.979} C_VEL
LIN {X 0,Y 587.164,Z 352.178,A -85,B 0,C 180,E1 -1367.016,E2 -1367.016} C_VEL
LIN {X 0,Y 587.165,Z 349.365,A -85,B 0,C 180,E1 -1367.77,E2 -1367.77} C_VEL
LIN {X 0,Y 587.215,Z 343.979,A -85,B 0,C 180,E1 -1368.852,E2 -1368.852} C_VEL
LIN {X 0,Y 587.22,Z 338.099,A -85,B 0,C 180,E1 -1369.76,E2 -1369.76} C_VEL
LIN {X 0,Y 587.278,Z 330.471,A -85,B 0,C 180,E1 -1370.672,E2 -1370.672} C_VEL
LIN {X 0,Y 587.314,Z 322.767,A -85,B 0,C 180,E1 -1371.405,E2 -1371.405} C_VEL
LIN {X 0,Y 587.323,Z 314.418,A -85,B 0,C 180,E1 -1372.05,E2 -1372.05} C_VEL
LIN {X 0,Y 587.423,Z 304.123,A -85,B 0,C 180,E1 -1372.68,E2 -1372.68} C_VEL
LIN {X 0,Y 587.455,Z 294.246,A -85,B 0,C 180,E1 -1373.132,E2 -1373.132} C_VEL
LIN {X 0,Y 587.492,Z 283.512,A -85,B 0,C 180,E1 -1373.484,E2 -1373.484} C_VEL
LIN {X 0,Y 587.133,Z 278.726,A -85,B 0,C 180,E1 -1373.616,E2 -1373.616} C_VEL
LIN {X 0,Y 587.108,Z 274.33,A -85,B 0,C 180,E1 -1376.288,E2 -1376.288} C_VEL
LIN {X 0,Y 587.143,Z 269.749,A -85,B 0,C 180,E1 -1379.102,E2 -1379.102} C_VEL
LIN {X 0,Y 587.147,Z 265.398,A -85,B 0,C 180,E1 -1381.809,E2 -1381.809} C_VEL
LIN {X 0,Y 587.123,Z 261.423,A -85,B 0,C 180,E1 -1384.319,E2 -1384.319} C_VEL
LIN {X 0,Y 587.125,Z 257.616,A -85,B 0,C 180,E1 -1386.762,E2 -1386.762} C_VEL
LIN {X 0,Y 587.171,Z 253.838,A -85,B 0,C 180,E1 -1389.372,E2 -1389.372} C_VEL
LIN {X 0,Y 587.199,Z 249.86,A -85,B 0,C 180,E1 -1392.096,E2 -1392.096} C_VEL
LIN {X 0,Y 587.243,Z 245.708,A -85,B 0,C 180,E1 -1394.917,E2 -1394.917} C_VEL
LIN {X 0,Y 587.245,Z 244.152,A -85,B 0,C 180,E1 -1396.045,E2 -1396.045} C_VEL
LIN {X 0,Y 587.331,Z 244.142,A -85,B 0,C 180,E1 -1397.928,E2 -1397.928} C_VEL
LIN {X 0,Y 587.318,Z 244.143,A -85,B 0,C 180,E1 -1401.058,E2 -1401.058} C_VEL
LIN {X 0,Y 587.337,Z 244.135,A -85,B 0,C 180,E1 -1403.292,E2 -1403.292} C_VEL
LIN {X 0,Y 587.351,Z 244.138,A -85,B 0,C 180,E1 -1405.782,E2 -1405.782} C_VEL
LIN {X 0,Y 587.322,Z 244.136,A -85,B 0,C 180,E1 -1408.232,E2 -1408.232} C_VEL
LIN {X 0,Y 587.339,Z 244.137,A -85,B 0,C 180,E1 -1410.866,E2 -1410.866} C_VEL
LIN {X 0,Y 587.341,Z 244.14,A -85,B 0,C 180,E1 -1413.82,E2 -1413.82} C_VEL
LIN {X 0,Y 587.304,Z 244.138,A -85,B 0,C 180,E1 -1415.994,E2 -1415.994} C_VEL
LIN {X 0,Y 587.341,Z 244.135,A -85,B 0,C 180,E1 -1418.956,E2 -1418.956} C_VEL
LIN {X 0,Y 587.316,Z 244.141,A -85,B 0,C 180,E1 -1421.875,E2 -1421.875} C_VEL
LIN {X 0,Y 587.305,Z 244.138,A -85,B 0,C 180,E1 -1424.026,E2 -1424.026} C_VEL
LIN {X 0,Y 587.308,Z 244.139,A -85,B 0,C 180,E1 -1426.86,E2 -1426.86} C_VEL
LIN {X 0,Y 587.335,Z 244.14,A -85,B 0,C 180,E1 -1429.661,E2 -1429.661} C_VEL
LIN {X 0,Y 587.349,Z 244.135,A -85,B 0,C 180,E1 -1432.438,E2 -1432.438} C_VEL
LIN {X 0,Y 587.346,Z 244.133,A -85,B 0,C 180,E1 -1435.197,E2 -1435.197} C_VEL
LIN {X 0,Y 587.358,Z 244.133,A -85,B 0,C 180,E1 -1437.944,E2 -1437.944} C_VEL
LIN {X 0,Y 587.39,Z 244.134,A -85,B 0,C 180,E1 -1440.687,E2 -1440.687} C_VEL
LIN {X 0,Y 587.31,Z 244.139,A -85,B 0,C 180,E1 -1443.431,E2 -1443.431} C_VEL
LIN {X 0,Y 587.353,Z 244.138,A -85,B 0,C 180,E1 -1445.494,E2 -1445.494} C_VEL
LIN {X 0,Y 587.359,Z 244.133,A -85,B 0,C 180,E1 -1448.256,E2 -1448.256} C_VEL
LIN {X 0,Y 587.338,Z 244.134,A -85,B 0,C 180,E1 -1451.135,E2 -1451.135} C_VEL
LIN {X 0,Y 587.357,Z 244.132,A -85,B 0,C 180,E1 -1454.262,E2 -1454.262} C_VEL
LIN {X 0,Y 587.336,Z 244.134,A -85,B 0,C 180,E1 -1457.407,E2 -1457.407} C_VEL
LIN {X 0,Y 587.313,Z 244.138,A -85,B 0,C 180,E1 -1460.306,E2 -1460.306} C_VEL
LIN {X 0,Y 587.319,Z 244.138,A -85,B 0,C 180,E1 -1463.26,E2 -1463.26} C_VEL
LIN {X 0,Y 587.327,Z 244.136,A -85,B 0,C 180,E1 -1465.518,E2 -1465.518} C_VEL
LIN {X 0,Y 587.295,Z 244.144,A -85,B 0,C 180,E1 -1467.821,E2 -1467.821} C_VEL
LIN {X 0,Y 587.336,Z 244.138,A -85,B 0,C 180,E1 -1470.512,E2 -1470.512} C_VEL
LIN {X 0,Y 587.335,Z 244.135,A -85,B 0,C 180,E1 -1473.113,E2 -1473.113} C_VEL
LIN {X 0,Y 587.285,Z 244.148,A -85,B 0,C 180,E1 -1475.538,E2 -1475.538} C_VEL
LIN {X 0,Y 587.325,Z 244.139,A -85,B 0,C 180,E1 -1478.48,E2 -1478.48} C_VEL
LIN {X 0,Y 587.333,Z 244.135,A -85,B 0,C 180,E1 -1481.158,E2 -1481.158} C_VEL
LIN {X 0,Y 587.305,Z 244.139,A -85,B 0,C 180,E1 -1484.113,E2 -1484.113} C_VEL
LIN {X 0,Y 587.311,Z 244.14,A -85,B 0,C 180,E1 -1486.995,E2 -1486.995} C_VEL
LIN {X 0,Y 587.319,Z 244.143,A -85,B 0,C 180,E1 -1489.748,E2 -1489.748} C_VEL
LIN {X 0,Y 587.334,Z 244.136,A -85,B 0,C 180,E1 -1492.393,E2 -1492.393} C_VEL
LIN {X 0,Y 587.344,Z 244.136,A -85,B 0,C 180,E1 -1495.653,E2 -1495.653} C_VEL
LIN {X 0,Y 587.393,Z 244.26,A -85,B 0,C 180,E1 -1496.829,E2 -1496.829} C_VEL
LIN {X 0,Y 587.555,Z 248.593,A -85,B 0,C 180,E1 -1498.245,E2 -1498.245} C_VEL
LIN {X 0,Y 587.515,Z 256.769,A -85,B 0,C 180,E1 -1500.838,E2 -1500.838} C_VEL
LIN {X 0,Y 587.456,Z 265.147,A -85,B 0,C 180,E1 -1503.345,E2 -1503.345} C_VEL
LIN {X 0,Y 587.367,Z 274.213,A -85,B 0,C 180,E1 -1505.996,E2 -1505.996} C_VEL
LIN {X 0,Y 587.329,Z 284.431,A -85,B 0,C 180,E1 -1508.964,E2 -1508.964} C_VEL
LIN {X 0,Y 587.268,Z 294.65,A -85,B 0,C 180,E1 -1511.873,E2 -1511.873} C_VEL
LIN {X 0,Y 587.241,Z 304.869,A -85,B 0,C 180,E1 -1514.736,E2 -1514.736} C_VEL
LIN {X 0,Y 587.226,Z 315.087,A -85,B 0,C 180,E1 -1517.56,E2 -1517.56} C_VEL
LIN {X 0,Y 587.199,Z 325.306,A -85,B 0,C 180,E1 -1520.355,E2 -1520.355} C_VEL
LIN {X 0,Y 587.495,Z 334.112,A -85,B 0,C 180,E1 -1520.577,E2 -1520.577} C_VEL
LIN {X 0,Y 587.441,Z 345.637,A -85,B 0,C 180,E1 -1520.967,E2 -1520.967} C_VEL
LIN {X 0,Y 587.371,Z 356.252,A -85,B 0,C 180,E1 -1521.486,E2 -1521.486} C_VEL
LIN {X 0,Y 587.359,Z 364.561,A -85,B 0,C 180,E1 -1522.005,E2 -1522.005} C_VEL
LIN {X 0,Y 587.296,Z 372.414,A -85,B 0,C 180,E1 -1522.61,E2 -1522.61} C_VEL
LIN {X 0,Y 587.294,Z 380.089,A -85,B 0,C 180,E1 -1523.335,E2 -1523.335} C_VEL
LIN {X 0,Y 587.253,Z 387.198,A -85,B 0,C 180,E1 -1524.162,E2 -1524.162} C_VEL
LIN {X 0,Y 587.203,Z 393.034,A -85,B 0,C 180,E1 -1525.023,E2 -1525.023} C_VEL
LIN {X 0,Y 587.181,Z 397.635,A -85,B 0,C 180,E1 -1525.883,E2 -1525.883} C_VEL
LIN {X 0,Y 587.191,Z 400.625,A -85,B 0,C 180,E1 -1526.57,E2 -1526.57} C_VEL
LIN {X 0,Y 587.135,Z 402.936,A -85,B 0,C 180,E1 -1527.257,E2 -1527.257} C_VEL
LIN {X 0,Y 587.141,Z 404.682,A -85,B 0,C 180,E1 -1527.943,E2 -1527.943} C_VEL
LIN {X 0,Y 587.145,Z 405.937,A -85,B 0,C 180,E1 -1528.629,E2 -1528.629} C_VEL
LIN {X 0,Y 587.136,Z 406.712,A -85,B 0,C 180,E1 -1529.315,E2 -1529.315} C_VEL
LIN {X 0,Y 587.134,Z 407,A -85,B 0,C 180,E1 -1530.001,E2 -1530.001} C_VEL
LIN {X 0,Y 587.136,Z 406.711,A -85,B 0,C 180,E1 -1530.687,E2 -1530.687} C_VEL
LIN {X 0,Y 587.145,Z 405.934,A -85,B 0,C 180,E1 -1531.373,E2 -1531.373} C_VEL
LIN {X 0,Y 587.141,Z 404.678,A -85,B 0,C 180,E1 -1532.059,E2 -1532.059} C_VEL
LIN {X 0,Y 587.155,Z 401.785,A -85,B 0,C 180,E1 -1533.088,E2 -1533.088} C_VEL
LIN {X 0,Y 587.21,Z 399.143,A -85,B 0,C 180,E1 -1533.775,E2 -1533.775} C_VEL
LIN {X 0,Y 587.17,Z 393.98,A -85,B 0,C 180,E1 -1534.807,E2 -1534.807} C_VEL
LIN {X 0,Y 587.253,Z 387.181,A -85,B 0,C 180,E1 -1535.839,E2 -1535.839} C_VEL
LIN {X 0,Y 587.27,Z 380.285,A -85,B 0,C 180,E1 -1536.646,E2 -1536.646} C_VEL
LIN {X 0,Y 587.293,Z 373.409,A -85,B 0,C 180,E1 -1537.306,E2 -1537.306} C_VEL
LIN {X 0,Y 587.347,Z 365.756,A -85,B 0,C 180,E1 -1537.91,E2 -1537.91} C_VEL
LIN {X 0,Y 587.378,Z 357.714,A -85,B 0,C 180,E1 -1538.429,E2 -1538.429} C_VEL
LIN {X 0,Y 587.404,Z 349.381,A -85,B 0,C 180,E1 -1538.862,E2 -1538.862} C_VEL
LIN {X 0,Y 587.465,Z 340.87,A -85,B 0,C 180,E1 -1539.208,E2 -1539.208} C_VEL
LIN {X 0,Y 587.492,Z 330.722,A -85,B 0,C 180,E1 -1539.512,E2 -1539.512} C_VEL
LIN {X 0,Y 587.199,Z 325.299,A -85,B 0,C 180,E1 -1539.647,E2 -1539.647} C_VEL
LIN {X 0,Y 587.228,Z 315.081,A -85,B 0,C 180,E1 -1542.441,E2 -1542.441} C_VEL
LIN {X 0,Y 587.243,Z 304.862,A -85,B 0,C 180,E1 -1545.266,E2 -1545.266} C_VEL
LIN {X 0,Y 587.266,Z 294.643,A -85,B 0,C 180,E1 -1548.129,E2 -1548.129} C_VEL
LIN {X 0,Y 587.313,Z 285.702,A -85,B 0,C 180,E1 -1550.672,E2 -1550.672} C_VEL
LIN {X 0,Y 587.392,Z 276.761,A -85,B 0,C 180,E1 -1553.257,E2 -1553.257} C_VEL
LIN {X 0,Y 587.441,Z 266.412,A -85,B 0,C 180,E1 -1556.274,E2 -1556.274} C_VEL
LIN {X 0,Y 587.507,Z 258.68,A -85,B 0,C 180,E1 -1558.588,E2 -1558.588} C_VEL
LIN {X 0,Y 587.577,Z 249.841,A -85,B 0,C 180,E1 -1561.353,E2 -1561.353} C_VEL
LIN {X 0,Y 587.607,Z 246.076,A -85,B 0,C 180,E1 -1562.563,E2 -1562.563} C_VEL
LIN {X 0,Y 587.353,Z 244.139,A -85,B 0,C 180,E1 -1563.267,E2 -1563.267} C_VEL
LIN {X 0,Y 587.296,Z 244.144,A -85,B 0,C 180,E1 -1565.9,E2 -1565.9} C_VEL
LIN {X 0,Y 587.335,Z 244.14,A -85,B 0,C 180,E1 -1568.48,E2 -1568.48} C_VEL
LIN {X 0,Y 587.343,Z 244.138,A -85,B 0,C 180,E1 -1571.157,E2 -1571.157} C_VEL
LIN {X 0,Y 587.318,Z 244.141,A -85,B 0,C 180,E1 -1574.112,E2 -1574.112} C_VEL
LIN {X 0,Y 587.32,Z 244.14,A -85,B 0,C 180,E1 -1576.993,E2 -1576.993} C_VEL
LIN {X 0,Y 587.317,Z 244.141,A -85,B 0,C 180,E1 -1579.745,E2 -1579.745} C_VEL
LIN {X 0,Y 587.347,Z 244.139,A -85,B 0,C 180,E1 -1582.392,E2 -1582.392} C_VEL
LIN {X 0,Y 587.364,Z 244.136,A -85,B 0,C 180,E1 -1585.779,E2 -1585.779} C_VEL
LIN {X 0,Y 587.348,Z 244.137,A -85,B 0,C 180,E1 -1588.231,E2 -1588.231} C_VEL
LIN {X 0,Y 587.354,Z 244.137,A -85,B 0,C 180,E1 -1590.867,E2 -1590.867} C_VEL
LIN {X 0,Y 587.368,Z 244.135,A -85,B 0,C 180,E1 -1593.818,E2 -1593.818} C_VEL
LIN {X 0,Y 587.337,Z 244.138,A -85,B 0,C 180,E1 -1595.993,E2 -1595.993} C_VEL
LIN {X 0,Y 587.33,Z 244.139,A -85,B 0,C 180,E1 -1598.225,E2 -1598.225} C_VEL
LIN {X 0,Y 587.352,Z 244.136,A -85,B 0,C 180,E1 -1601.15,E2 -1601.15} C_VEL
LIN {X 0,Y 587.327,Z 244.14,A -85,B 0,C 180,E1 -1604.024,E2 -1604.024} C_VEL
LIN {X 0,Y 587.321,Z 244.142,A -85,B 0,C 180,E1 -1606.857,E2 -1606.857} C_VEL
LIN {X 0,Y 587.339,Z 244.139,A -85,B 0,C 180,E1 -1609.659,E2 -1609.659} C_VEL
LIN {X 0,Y 587.368,Z 244.134,A -85,B 0,C 180,E1 -1612.436,E2 -1612.436} C_VEL
LIN {X 0,Y 587.366,Z 244.135,A -85,B 0,C 180,E1 -1615.194,E2 -1615.194} C_VEL
LIN {X 0,Y 587.37,Z 244.137,A -85,B 0,C 180,E1 -1617.942,E2 -1617.942} C_VEL
LIN {X 0,Y 587.392,Z 244.132,A -85,B 0,C 180,E1 -1620.684,E2 -1620.684} C_VEL
LIN {X 0,Y 587.34,Z 244.137,A -85,B 0,C 180,E1 -1623.429,E2 -1623.429} C_VEL
LIN {X 0,Y 587.327,Z 244.141,A -85,B 0,C 180,E1 -1626.181,E2 -1626.181} C_VEL
LIN {X 0,Y 587.368,Z 244.135,A -85,B 0,C 180,E1 -1628.254,E2 -1628.254} C_VEL
LIN {X 0,Y 587.351,Z 244.138,A -85,B 0,C 180,E1 -1631.132,E2 -1631.132} C_VEL
LIN {X 0,Y 587.367,Z 244.136,A -85,B 0,C 180,E1 -1634.259,E2 -1634.259} C_VEL
LIN {X 0,Y 587.348,Z 244.137,A -85,B 0,C 180,E1 -1637.404,E2 -1637.404} C_VEL
LIN {X 0,Y 587.311,Z 244.143,A -85,B 0,C 180,E1 -1638.3,E2 -1638.3} C_VEL
LIN {X 0,Y 586.667,Z 244.223,A -85,B 0,C 180,E1 -1638.872,E2 -1638.872} C_VEL
LIN {X 0,Y 583.842,Z 244.576,A -85,B 0,C 180,E1 -1639.8,E2 -1639.8} C_VEL
LIN {X 0,Y 581.432,Z 244.878,A -85,B 0,C 180,E1 -1640.547,E2 -1640.547} C_VEL
LIN {X 0,Y 580.378,Z 245.008,A -85,B 0,C 180,E1 -1641.124,E2 -1641.124} C_VEL
LIN {X 0,Y 580.283,Z 245.018,A -85,B 0,C 180,E1 -1641.319,E2 -1641.319} C_VEL
LIN {X 0,Y 580.279,Z 245.018,A -85,B 0,C 180,E1 -1643.556,E2 -1643.556} C_VEL
LIN {X 0,Y 580.29,Z 245.016,A -85,B 0,C 180,E1 -1645.847,E2 -1645.847} C_VEL
LIN {X 0,Y 580.3,Z 245.017,A -85,B 0,C 180,E1 -1648.183,E2 -1648.183} C_VEL
LIN {X 0,Y 580.29,Z 245.016,A -85,B 0,C 180,E1 -1650.694,E2 -1650.694} C_VEL
LIN {X 0,Y 580.301,Z 245.017,A -85,B 0,C 180,E1 -1653.315,E2 -1653.315} C_VEL
LIN {X 0,Y 580.32,Z 245.012,A -85,B 0,C 180,E1 -1655.766,E2 -1655.766} C_VEL
LIN {X 0,Y 580.282,Z 245.018,A -85,B 0,C 180,E1 -1658.144,E2 -1658.144} C_VEL
LIN {X 0,Y 580.294,Z 245.016,A -85,B 0,C 180,E1 -1660.841,E2 -1660.841} C_VEL
LIN {X 0,Y 580.282,Z 245.018,A -85,B 0,C 180,E1 -1663.655,E2 -1663.655} C_VEL
LIN {X 0,Y 580.282,Z 245.019,A -85,B 0,C 180,E1 -1666.606,E2 -1666.606} C_VEL
LIN {X 0,Y 580.31,Z 245.014,A -85,B 0,C 180,E1 -1669.157,E2 -1669.157} C_VEL
LIN {X 0,Y 580.282,Z 245.017,A -85,B 0,C 180,E1 -1671.925,E2 -1671.925} C_VEL
LIN {X 0,Y 580.297,Z 245.017,A -85,B 0,C 180,E1 -1674.455,E2 -1674.455} C_VEL
LIN {X 0,Y 580.286,Z 245.017,A -85,B 0,C 180,E1 -1676.974,E2 -1676.974} C_VEL
LIN {X 0,Y 580.298,Z 245.016,A -85,B 0,C 180,E1 -1679.424,E2 -1679.424} C_VEL
LIN {X 0,Y 580.307,Z 245.014,A -85,B 0,C 180,E1 -1682.135,E2 -1682.135} C_VEL
LIN {X 0,Y 580.295,Z 245.016,A -85,B 0,C 180,E1 -1684.919,E2 -1684.919} C_VEL
LIN {X 0,Y 580.315,Z 245.013,A -85,B 0,C 180,E1 -1687.198,E2 -1687.198} C_VEL
LIN {X 0,Y 580.297,Z 245.015,A -85,B 0,C 180,E1 -1690.177,E2 -1690.177} C_VEL
LIN {X 0,Y 580.164,Z 245.202,A -85,B 0,C 180,E1 -1692.371,E2 -1692.371} C_VEL
LIN {X 0,Y 580.158,Z 249.367,A -85,B 0,C 180,E1 -1695.262,E2 -1695.262} C_VEL
LIN {X 0,Y 580.15,Z 253.494,A -85,B 0,C 180,E1 -1698.115,E2 -1698.115} C_VEL
LIN {X 0,Y 580.135,Z 257.578,A -85,B 0,C 180,E1 -1700.938,E2 -1700.938} C_VEL
LIN {X 0,Y 580.123,Z 261.771,A -85,B 0,C 180,E1 -1703.74,E2 -1703.74} C_VEL
LIN {X 0,Y 580.083,Z 266.137,A -85,B 0,C 180,E1 -1706.526,E2 -1706.526} C_VEL
LIN {X 0,Y 580.091,Z 270.555,A -85,B 0,C 180,E1 -1709.305,E2 -1709.305} C_VEL
LIN {X 0,Y 580.003,Z 275.031,A -85,B 0,C 180,E1 -1712.082,E2 -1712.082} C_VEL
LIN {X 0,Y 580.057,Z 278.702,A -85,B 0,C 180,E1 -1714.342,E2 -1714.342} C_VEL
LIN {X 0,Y 580.481,Z 285.147,A -85,B 0,C 180,E1 -1714.534,E2 -1714.534} C_VEL
LIN {X 0,Y 580.375,Z 296.696,A -85,B 0,C 180,E1 -1714.949,E2 -1714.949} C_VEL
LIN {X 0,Y 580.3,Z 307.027,A -85,B 0,C 180,E1 -1715.472,E2 -1715.472} C_VEL
LIN {X 0,Y 580.215,Z 315.186,A -85,B 0,C 180,E1 -1715.996,E2 -1715.996} C_VEL
LIN {X 0,Y 580.244,Z 322.893,A -85,B 0,C 180,E1 -1716.606,E2 -1716.606} C_VEL
LIN {X 0,Y 580.198,Z 330.168,A -85,B 0,C 180,E1 -1717.306,E2 -1717.306} C_VEL
LIN {X 0,Y 580.162,Z 337.545,A -85,B 0,C 180,E1 -1718.182,E2 -1718.182} C_VEL
LIN {X 0,Y 580.101,Z 343.328,A -85,B 0,C 180,E1 -1719.061,E2 -1719.061} C_VEL
LIN {X 0,Y 580.094,Z 347.134,A -85,B 0,C 180,E1 -1719.764,E2 -1719.764} C_VEL
LIN {X 0,Y 580.09,Z 351.335,A -85,B 0,C 180,E1 -1720.783,E2 -1720.783} C_VEL
LIN {X 0,Y 580.061,Z 354.504,A -85,B 0,C 180,E1 -1721.885,E2 -1721.885} C_VEL
LIN {X 0,Y 580.046,Z 355.852,A -85,B 0,C 180,E1 -1722.596,E2 -1722.596} C_VEL
LIN {X 0,Y 580.052,Z 356.691,A -85,B 0,C 180,E1 -1723.308,E2 -1723.308} C_VEL
LIN {X 0,Y 580.044,Z 356.936,A -85,B 0,C 180,E1 -1724.243,E2 -1724.243} C_VEL
LIN {X 0,Y 580.053,Z 355.902,A -85,B 0,C 180,E1 -1725.458,E2 -1725.458} C_VEL
LIN {X 0,Y 580.062,Z 354.562,A -85,B 0,C 180,E1 -1726.18,E2 -1726.18} C_VEL
LIN {X 0,Y 580.058,Z 351.469,A -85,B 0,C 180,E1 -1727.267,E2 -1727.267} C_VEL
LIN {X 0,Y 580.094,Z 346.973,A -85,B 0,C 180,E1 -1728.36,E2 -1728.36} C_VEL
LIN {X 0,Y 580.161,Z 342.827,A -85,B 0,C 180,E1 -1729.119,E2 -1729.119} C_VEL
LIN {X 0,Y 580.159,Z 336.744,A -85,B 0,C 180,E1 -1730.011,E2 -1730.011} C_VEL
LIN {X 0,Y 580.21,Z 330.706,A -85,B 0,C 180,E1 -1730.729,E2 -1730.729} C_VEL
LIN {X 0,Y 580.259,Z 322.805,A -85,B 0,C 180,E1 -1731.492,E2 -1731.492} C_VEL
LIN {X 0,Y 580.269,Z 315.765,A -85,B 0,C 180,E1 -1732.052,E2 -1732.052} C_VEL
LIN {X 0,Y 580.331,Z 308.725,A -85,B 0,C 180,E1 -1732.518,E2 -1732.518} C_VEL
LIN {X 0,Y 580.412,Z 300.713,A -85,B 0,C 180,E1 -1732.952,E2 -1732.952} C_VEL
LIN {X 0,Y 580.452,Z 291.367,A -85,B 0,C 180,E1 -1733.347,E2 -1733.347} C_VEL
LIN {X 0,Y 580.475,Z 282.294,A -85,B 0,C 180,E1 -1733.631,E2 -1733.631} C_VEL
LIN {X 0,Y 580.036,Z 278.727,A -85,B 0,C 180,E1 -1733.733,E2 -1733.733} C_VEL
LIN {X 0,Y 580.029,Z 274.016,A -85,B 0,C 180,E1 -1736.634,E2 -1736.634} C_VEL
LIN {X 0,Y 580.057,Z 269.779,A -85,B 0,C 180,E1 -1739.271,E2 -1739.271} C_VEL
LIN {X 0,Y 580.047,Z 265.113,A -85,B 0,C 180,E1 -1742.215,E2 -1742.215} C_VEL
LIN {X 0,Y 580.026,Z 261.215,A -85,B 0,C 180,E1 -1744.713,E2 -1744.713} C_VEL
LIN {X 0,Y 580.056,Z 257.432,A -85,B 0,C 180,E1 -1747.285,E2 -1747.285} C_VEL
LIN {X 0,Y 580.098,Z 253.2,A -85,B 0,C 180,E1 -1750.251,E2 -1750.251} C_VEL
LIN {X 0,Y 580.143,Z 249.57,A -85,B 0,C 180,E1 -1752.717,E2 -1752.717} C_VEL
LIN {X 0,Y 580.18,Z 245.39,A -85,B 0,C 180,E1 -1755.616,E2 -1755.616} C_VEL
LIN {X 0,Y 580.22,Z 245.024,A -85,B 0,C 180,E1 -1756.613,E2 -1756.613} C_VEL
LIN {X 0,Y 580.28,Z 245.015,A -85,B 0,C 180,E1 -1759.158,E2 -1759.158} C_VEL
LIN {X 0,Y 580.273,Z 245.014,A -85,B 0,C 180,E1 -1761.927,E2 -1761.927} C_VEL
LIN {X 0,Y 580.291,Z 245.016,A -85,B 0,C 180,E1 -1764.458,E2 -1764.458} C_VEL
LIN {X 0,Y 580.271,Z 245.016,A -85,B 0,C 180,E1 -1766.976,E2 -1766.976} C_VEL
LIN {X 0,Y 580.278,Z 245.015,A -85,B 0,C 180,E1 -1769.426,E2 -1769.426} C_VEL
LIN {X 0,Y 580.303,Z 245.016,A -85,B 0,C 180,E1 -1772.138,E2 -1772.138} C_VEL
LIN {X 0,Y 580.302,Z 245.016,A -85,B 0,C 180,E1 -1775.271,E2 -1775.271} C_VEL
LIN {X 0,Y 580.258,Z 245.017,A -85,B 0,C 180,E1 -1777.949,E2 -1777.949} C_VEL
LIN {X 0,Y 580.302,Z 245.01,A -85,B 0,C 180,E1 -1780.915,E2 -1780.915} C_VEL
LIN {X 0,Y 580.26,Z 245.016,A -85,B 0,C 180,E1 -1783.827,E2 -1783.827} C_VEL
LIN {X 0,Y 580.262,Z 245.019,A -85,B 0,C 180,E1 -1786.697,E2 -1786.697} C_VEL
LIN {X 0,Y 580.318,Z 245.008,A -85,B 0,C 180,E1 -1788.829,E2 -1788.829} C_VEL
LIN {X 0,Y 580.293,Z 245.013,A -85,B 0,C 180,E1 -1791.645,E2 -1791.645} C_VEL
LIN {X 0,Y 580.311,Z 245.015,A -85,B 0,C 180,E1 -1794.441,E2 -1794.441} C_VEL
LIN {X 0,Y 580.339,Z 245.008,A -85,B 0,C 180,E1 -1797.225,E2 -1797.225} C_VEL
LIN {X 0,Y 580.332,Z 245.007,A -85,B 0,C 180,E1 -1800.001,E2 -1800.001} C_VEL
LIN {X 0,Y 580.328,Z 245.008,A -85,B 0,C 180,E1 -1802.778,E2 -1802.778} C_VEL
LIN {X 0,Y 580.319,Z 245.013,A -85,B 0,C 180,E1 -1805.561,E2 -1805.561} C_VEL
LIN {X 0,Y 580.323,Z 245.011,A -85,B 0,C 180,E1 -1808.357,E2 -1808.357} C_VEL
LIN {X 0,Y 580.29,Z 245.012,A -85,B 0,C 180,E1 -1811.192,E2 -1811.192} C_VEL
LIN {X 0,Y 580.319,Z 245.009,A -85,B 0,C 180,E1 -1814.018,E2 -1814.018} C_VEL
LIN {X 0,Y 580.303,Z 245.012,A -85,B 0,C 180,E1 -1816.915,E2 -1816.915} C_VEL
LIN {X 0,Y 580.275,Z 245.019,A -85,B 0,C 180,E1 -1819.824,E2 -1819.824} C_VEL
LIN {X 0,Y 580.268,Z 245.015,A -85,B 0,C 180,E1 -1822.054,E2 -1822.054} C_VEL
LIN {X 0,Y 580.299,Z 245.011,A -85,B 0,C 180,E1 -1825.081,E2 -1825.081} C_VEL
LIN {X 0,Y 580.27,Z 245.016,A -85,B 0,C 180,E1 -1828.188,E2 -1828.188} C_VEL
LIN {X 0,Y 580.287,Z 245.018,A -85,B 0,C 180,E1 -1830.698,E2 -1830.698} C_VEL
LIN {X 0,Y 580.3,Z 245.012,A -85,B 0,C 180,E1 -1833.318,E2 -1833.318} C_VEL
LIN {X 0,Y 580.234,Z 245.023,A -85,B 0,C 180,E1 -1835.757,E2 -1835.757} C_VEL
LIN {X 0,Y 580.281,Z 245.014,A -85,B 0,C 180,E1 -1838.148,E2 -1838.148} C_VEL
LIN {X 0,Y 580.296,Z 245.012,A -85,B 0,C 180,E1 -1840.844,E2 -1840.844} C_VEL
LIN {X 0,Y 580.266,Z 245.02,A -85,B 0,C 180,E1 -1843.66,E2 -1843.66} C_VEL
LIN {X 0,Y 580.27,Z 245.021,A -85,B 0,C 180,E1 -1846.611,E2 -1846.611} C_VEL
LIN {X 0,Y 580.3,Z 245.012,A -85,B 0,C 180,E1 -1849.158,E2 -1849.158} C_VEL
LIN {X 0,Y 580.279,Z 245.015,A -85,B 0,C 180,E1 -1851.929,E2 -1851.929} C_VEL
LIN {X 0,Y 580.246,Z 245.024,A -85,B 0,C 180,E1 -1854.454,E2 -1854.454} C_VEL
LIN {X 0,Y 580.362,Z 245.146,A -85,B 0,C 180,E1 -1856.676,E2 -1856.676} C_VEL
LIN {X 0,Y 580.579,Z 248.932,A -85,B 0,C 180,E1 -1857.926,E2 -1857.926} C_VEL
LIN {X 0,Y 580.53,Z 257.398,A -85,B 0,C 180,E1 -1860.651,E2 -1860.651} C_VEL
LIN {X 0,Y 580.422,Z 266.278,A -85,B 0,C 180,E1 -1863.385,E2 -1863.385} C_VEL
LIN {X 0,Y 580.346,Z 275.439,A -85,B 0,C 180,E1 -1866.067,E2 -1866.067} C_VEL
LIN {X 0,Y 580.302,Z 284.907,A -85,B 0,C 180,E1 -1868.835,E2 -1868.835} C_VEL
LIN {X 0,Y 580.212,Z 294.65,A -85,B 0,C 180,E1 -1871.644,E2 -1871.644} C_VEL
LIN {X 0,Y 580.184,Z 303.591,A -85,B 0,C 180,E1 -1874.185,E2 -1874.185} C_VEL
LIN {X 0,Y 580.163,Z 312.533,A -85,B 0,C 180,E1 -1876.694,E2 -1876.694} C_VEL
LIN {X 0,Y 580.148,Z 321.575,A -85,B 0,C 180,E1 -1879.206,E2 -1879.206} C_VEL
LIN {X 0,Y 580.118,Z 325.306,A -85,B 0,C 180,E1 -1880.236,E2 -1880.236} C_VEL
LIN {X 0,Y 580.511,Z 332.451,A -85,B 0,C 180,E1 -1880.419,E2 -1880.419} C_VEL
LIN {X 0,Y 580.441,Z 340.92,A -85,B 0,C 180,E1 -1880.681,E2 -1880.681} C_VEL
LIN {X 0,Y 580.393,Z 349.422,A -85,B 0,C 180,E1 -1881.032,E2 -1881.032} C_VEL
LIN {X 0,Y 580.341,Z 357.747,A -85,B 0,C 180,E1 -1881.47,E2 -1881.47} C_VEL
LIN {X 0,Y 580.299,Z 365.781,A -85,B 0,C 180,E1 -1881.995,E2 -1881.995} C_VEL
LIN {X 0,Y 580.225,Z 374.441,A -85,B 0,C 180,E1 -1882.694,E2 -1882.694} C_VEL
LIN {X 0,Y 580.218,Z 382.426,A -85,B 0,C 180,E1 -1883.504,E2 -1883.504} C_VEL
LIN {X 0,Y 580.173,Z 388.439,A -85,B 0,C 180,E1 -1884.265,E2 -1884.265} C_VEL
LIN {X 0,Y 580.084,Z 393.992,A -85,B 0,C 180,E1 -1885.136,E2 -1885.136} C_VEL
LIN {X 0,Y 580.122,Z 399.152,A -85,B 0,C 180,E1 -1886.18,E2 -1886.18} C_VEL
LIN {X 0,Y 580.07,Z 401.792,A -85,B 0,C 180,E1 -1886.876,E2 -1886.876} C_VEL
LIN {X 0,Y 580.04,Z 404.683,A -85,B 0,C 180,E1 -1887.918,E2 -1887.918} C_VEL
LIN {X 0,Y 580.045,Z 405.938,A -85,B 0,C 180,E1 -1888.612,E2 -1888.612} C_VEL
LIN {X 0,Y 580.036,Z 406.711,A -85,B 0,C 180,E1 -1889.307,E2 -1889.307} C_VEL
LIN {X 0,Y 580.034,Z 407,A -85,B 0,C 180,E1 -1890.001,E2 -1890.001} C_VEL
LIN {X 0,Y 580.036,Z 406.71,A -85,B 0,C 180,E1 -1890.695,E2 -1890.695} C_VEL
LIN {X 0,Y 580.045,Z 405.935,A -85,B 0,C 180,E1 -1891.389,E2 -1891.389} C_VEL
LIN {X 0,Y 580.04,Z 404.678,A -85,B 0,C 180,E1 -1892.084,E2 -1892.084} C_VEL
LIN {X 0,Y 580.07,Z 401.785,A -85,B 0,C 180,E1 -1893.126,E2 -1893.126} C_VEL
LIN {X 0,Y 580.122,Z 399.144,A -85,B 0,C 180,E1 -1893.821,E2 -1893.821} C_VEL
LIN {X 0,Y 580.084,Z 393.981,A -85,B 0,C 180,E1 -1894.866,E2 -1894.866} C_VEL
LIN {X 0,Y 580.194,Z 387.18,A -85,B 0,C 180,E1 -1895.911,E2 -1895.911} C_VEL
LIN {X 0,Y 580.227,Z 379.493,A -85,B 0,C 180,E1 -1896.808,E2 -1896.808} C_VEL
LIN {X 0,Y 580.255,Z 372.396,A -85,B 0,C 180,E1 -1897.482,E2 -1897.482} C_VEL
LIN {X 0,Y 580.322,Z 364.535,A -85,B 0,C 180,E1 -1898.094,E2 -1898.094} C_VEL
LIN {X 0,Y 580.39,Z 354.718,A -85,B 0,C 180,E1 -1898.707,E2 -1898.707} C_VEL
LIN {X 0,Y 580.462,Z 343.278,A -85,B 0,C 180,E1 -1899.232,E2 -1899.232} C_VEL
LIN {X 0,Y 580.501,Z 334.044,A -85,B 0,C 180,E1 -1899.539,E2 -1899.539} C_VEL
LIN {X 0,Y 580.299,Z 326.988,A -85,B 0,C 180,E1 -1899.719,E2 -1899.719} C_VEL
LIN {X 0,Y 580.118,Z 325.299,A -85,B 0,C 180,E1 -1899.766,E2 -1899.766} C_VEL
LIN {X 0,Y 580.168,Z 315.081,A -85,B 0,C 180,E1 -1902.595,E2 -1902.595} C_VEL
LIN {X 0,Y 580.181,Z 304.862,A -85,B 0,C 180,E1 -1905.457,E2 -1905.457} C_VEL
LIN {X 0,Y 580.207,Z 294.643,A -85,B 0,C 180,E1 -1908.358,E2 -1908.358} C_VEL
LIN {X 0,Y 580.308,Z 284.9,A -85,B 0,C 180,E1 -1911.167,E2 -1911.167} C_VEL
LIN {X 0,Y 580.347,Z 275.404,A -85,B 0,C 180,E1 -1913.935,E2 -1913.935} C_VEL
LIN {X 0,Y 580.415,Z 266.303,A -85,B 0,C 180,E1 -1916.617,E2 -1916.617} C_VEL
LIN {X 0,Y 580.5,Z 258.648,A -85,B 0,C 180,E1 -1918.966,E2 -1918.966} C_VEL
LIN {X 0,Y 580.582,Z 249.986,A -85,B 0,C 180,E1 -1921.721,E2 -1921.721} C_VEL
LIN {X 0,Y 580.487,Z 246.072,A -85,B 0,C 180,E1 -1923.013,E2 -1923.013} C_VEL
LIN {X 0,Y 580.331,Z 245.014,A -85,B 0,C 180,E1 -1923.404,E2 -1923.404} C_VEL
LIN {X 0,Y 580.274,Z 245.02,A -85,B 0,C 180,E1 -1926.404,E2 -1926.404} C_VEL
LIN {X 0,Y 580.303,Z 245.016,A -85,B 0,C 180,E1 -1929.186,E2 -1929.186} C_VEL
LIN {X 0,Y 580.287,Z 245.017,A -85,B 0,C 180,E1 -1931.769,E2 -1931.769} C_VEL
LIN {X 0,Y 580.255,Z 245.021,A -85,B 0,C 180,E1 -1934.628,E2 -1934.628} C_VEL
LIN {X 0,Y 580.293,Z 245.017,A -85,B 0,C 180,E1 -1937.628,E2 -1937.628} C_VEL
LIN {X 0,Y 580.289,Z 245.016,A -85,B 0,C 180,E1 -1940.066,E2 -1940.066} C_VEL
LIN {X 0,Y 580.284,Z 245.017,A -85,B 0,C 180,E1 -1943.068,E2 -1943.068} C_VEL
LIN {X 0,Y 580.321,Z 245.012,A -85,B 0,C 180,E1 -1946.145,E2 -1946.145} C_VEL
LIN {X 0,Y 580.283,Z 245.019,A -85,B 0,C 180,E1 -1948.614,E2 -1948.614} C_VEL
LIN {X 0,Y 580.297,Z 245.015,A -85,B 0,C 180,E1 -1951.023,E2 -1951.023} C_VEL
LIN {X 0,Y 580.3,Z 245.017,A -85,B 0,C 180,E1 -1953.666,E2 -1953.666} C_VEL
LIN {X 0,Y 580.306,Z 245.016,A -85,B 0,C 180,E1 -1955.683,E2 -1955.683} C_VEL
LIN {X 0,Y 580.293,Z 245.018,A -85,B 0,C 180,E1 -1958.694,E2 -1958.694} C_VEL
LIN {X 0,Y 580.303,Z 245.016,A -85,B 0,C 180,E1 -1960.913,E2 -1960.913} C_VEL
LIN {X 0,Y 580.277,Z 245.019,A -85,B 0,C 180,E1 -1963.825,E2 -1963.825} C_VEL
LIN {X 0,Y 580.278,Z 245.019,A -85,B 0,C 180,E1 -1966.695,E2 -1966.695} C_VEL
LIN {X 0,Y 580.313,Z 245.016,A -85,B 0,C 180,E1 -1968.826,E2 -1968.826} C_VEL
LIN {X 0,Y 580.316,Z 245.014,A -85,B 0,C 180,E1 -1971.643,E2 -1971.643} C_VEL
LIN {X 0,Y 580.28,Z 245.019,A -85,B 0,C 180,E1 -1973.741,E2 -1973.741} C_VEL
LIN {X 0,Y 580.273,Z 245.02,A -85,B 0,C 180,E1 -1975.832,E2 -1975.832} C_VEL
LIN {X 0,Y 580.342,Z 245.012,A -85,B 0,C 180,E1 -1977.917,E2 -1977.917} C_VEL
LIN {X 0,Y 580.364,Z 245.008,A -85,B 0,C 180,E1 -1980.693,E2 -1980.693} C_VEL
LIN {X 0,Y 580.291,Z 245.015,A -85,B 0,C 180,E1 -1983.47,E2 -1983.47} C_VEL
LIN {X 0,Y 580.331,Z 245.01,A -85,B 0,C 180,E1 -1985.558,E2 -1985.558} C_VEL
LIN {X 0,Y 580.331,Z 245.011,A -85,B 0,C 180,E1 -1988.355,E2 -1988.355} C_VEL
LIN {X 0,Y 580.303,Z 245.016,A -85,B 0,C 180,E1 -1991.189,E2 -1991.189} C_VEL
LIN {X 0,Y 580.328,Z 245.013,A -85,B 0,C 180,E1 -1994.015,E2 -1994.015} C_VEL
LIN {X 0,Y 580.313,Z 245.014,A -85,B 0,C 180,E1 -1996.912,E2 -1996.912} C_VEL
LIN {X 0,Y 580.306,Z 245.014,A -85,B 0,C 180,E1 -1999.821,E2 -1999.821} C_VEL
LIN {X 0,Y 580.283,Z 245.018,A -85,B 0,C 180,E1 -2001.319,E2 -2001.319} C_VEL
LIN {X 0,Y 579.586,Z 245.105,A -85,B 0,C 180,E1 -2001.898,E2 -2001.898} C_VEL
LIN {X 0,Y 576.71,Z 245.462,A -85,B 0,C 180,E1 -2002.838,E2 -2002.838} C_VEL
LIN {X 0,Y 574.315,Z 245.761,A -85,B 0,C 180,E1 -2003.595,E2 -2003.595} C_VEL
LIN {X 0,Y 573.315,Z 245.887,A -85,B 0,C 180,E1 -2004.178,E2 -2004.178} C_VEL
LIN {X 0,Y 573.248,Z 245.892,A -85,B 0,C 180,E1 -2004.376,E2 -2004.376} C_VEL
LIN {X 0,Y 573.25,Z 245.893,A -85,B 0,C 180,E1 -2006.974,E2 -2006.974} C_VEL
LIN {X 0,Y 573.245,Z 245.895,A -85,B 0,C 180,E1 -2009.487,E2 -2009.487} C_VEL
LIN {X 0,Y 573.254,Z 245.895,A -85,B 0,C 180,E1 -2012.227,E2 -2012.227} C_VEL
LIN {X 0,Y 573.246,Z 245.893,A -85,B 0,C 180,E1 -2014.772,E2 -2014.772} C_VEL
LIN {X 0,Y 573.248,Z 245.894,A -85,B 0,C 180,E1 -2017.164,E2 -2017.164} C_VEL
LIN {X 0,Y 573.241,Z 245.895,A -85,B 0,C 180,E1 -2019.605,E2 -2019.605} C_VEL
LIN {X 0,Y 573.243,Z 245.895,A -85,B 0,C 180,E1 -2022.641,E2 -2022.641} C_VEL
LIN {X 0,Y 573.229,Z 245.896,A -85,B 0,C 180,E1 -2025.665,E2 -2025.665} C_VEL
LIN {X 0,Y 573.251,Z 245.895,A -85,B 0,C 180,E1 -2028.544,E2 -2028.544} C_VEL
LIN {X 0,Y 573.24,Z 245.895,A -85,B 0,C 180,E1 -2031.297,E2 -2031.297} C_VEL
LIN {X 0,Y 573.253,Z 245.892,A -85,B 0,C 180,E1 -2034.009,E2 -2034.009} C_VEL
LIN {X 0,Y 573.271,Z 245.892,A -85,B 0,C 180,E1 -2036.517,E2 -2036.517} C_VEL
LIN {X 0,Y 573.233,Z 245.895,A -85,B 0,C 180,E1 -2039.113,E2 -2039.113} C_VEL
LIN {X 0,Y 573.252,Z 245.893,A -85,B 0,C 180,E1 -2041.966,E2 -2041.966} C_VEL
LIN {X 0,Y 573.244,Z 245.896,A -85,B 0,C 180,E1 -2044.589,E2 -2044.589} C_VEL
LIN {X 0,Y 573.246,Z 245.895,A -85,B 0,C 180,E1 -2047.662,E2 -2047.662} C_VEL
LIN {X 0,Y 573.26,Z 245.894,A -85,B 0,C 180,E1 -2050.669,E2 -2050.669} C_VEL
LIN {X 0,Y 573.118,Z 245.912,A -85,B 0,C 180,E1 -2052.147,E2 -2052.147} C_VEL
LIN {X 0,Y 573.101,Z 247.657,A -85,B 0,C 180,E1 -2053.617,E2 -2053.617} C_VEL
LIN {X 0,Y 573.084,Z 251.826,A -85,B 0,C 180,E1 -2056.525,E2 -2056.525} C_VEL
LIN {X 0,Y 573.088,Z 255.139,A -85,B 0,C 180,E1 -2058.822,E2 -2058.822} C_VEL
LIN {X 0,Y 573.048,Z 259.034,A -85,B 0,C 180,E1 -2061.536,E2 -2061.536} C_VEL
LIN {X 0,Y 573.062,Z 262.11,A -85,B 0,C 180,E1 -2063.662,E2 -2063.662} C_VEL
LIN {X 0,Y 573.012,Z 266.418,A -85,B 0,C 180,E1 -2066.483,E2 -2066.483} C_VEL
LIN {X 0,Y 572.997,Z 270.836,A -85,B 0,C 180,E1 -2069.296,E2 -2069.296} C_VEL
LIN {X 0,Y 572.907,Z 275.312,A -85,B 0,C 180,E1 -2072.108,E2 -2072.108} C_VEL
LIN {X 0,Y 572.972,Z 278.908,A -85,B 0,C 180,E1 -2074.242,E2 -2074.242} C_VEL
LIN {X 0,Y 573.489,Z 285.833,A -85,B 0,C 180,E1 -2074.436,E2 -2074.436} C_VEL
LIN {X 0,Y 573.354,Z 296.628,A -85,B 0,C 180,E1 -2074.833,E2 -2074.833} C_VEL
LIN {X 0,Y 573.276,Z 306.969,A -85,B 0,C 180,E1 -2075.363,E2 -2075.363} C_VEL
LIN {X 0,Y 573.165,Z 315.143,A -85,B 0,C 180,E1 -2075.893,E2 -2075.893} C_VEL
LIN {X 0,Y 573.197,Z 322.805,A -85,B 0,C 180,E1 -2076.506,E2 -2076.506} C_VEL
LIN {X 0,Y 573.127,Z 330.14,A -85,B 0,C 180,E1 -2077.22,E2 -2077.22} C_VEL
LIN {X 0,Y 573.105,Z 337.518,A -85,B 0,C 180,E1 -2078.106,E2 -2078.106} C_VEL
LIN {X 0,Y 573.022,Z 343.311,A -85,B 0,C 180,E1 -2078.996,E2 -2078.996} C_VEL
LIN {X 0,Y 573.008,Z 347.896,A -85,B 0,C 180,E1 -2079.886,E2 -2079.886} C_VEL
LIN {X 0,Y 573.009,Z 350.87,A -85,B 0,C 180,E1 -2080.6,E2 -2080.6} C_VEL
LIN {X 0,Y 572.99,Z 353.201,A -85,B 0,C 180,E1 -2081.317,E2 -2081.317} C_VEL
LIN {X 0,Y 572.979,Z 354.904,A -85,B 0,C 180,E1 -2082.034,E2 -2082.034} C_VEL
LIN {X 0,Y 572.941,Z 356.092,A -85,B 0,C 180,E1 -2082.755,E2 -2082.755} C_VEL
LIN {X 0,Y 572.959,Z 356.771,A -85,B 0,C 180,E1 -2083.476,E2 -2083.476} C_VEL
LIN {X 0,Y 572.957,Z 356.909,A -85,B 0,C 180,E1 -2084.307,E2 -2084.307} C_VEL
LIN {X 0,Y 572.948,Z 356.609,A -85,B 0,C 180,E1 -2084.926,E2 -2084.926} C_VEL
LIN {X 0,Y 572.948,Z 355.655,A -85,B 0,C 180,E1 -2085.655,E2 -2085.655} C_VEL
LIN {X 0,Y 573.006,Z 352.683,A -85,B 0,C 180,E1 -2086.934,E2 -2086.934} C_VEL
LIN {X 0,Y 572.986,Z 349.396,A -85,B 0,C 180,E1 -2087.856,E2 -2087.856} C_VEL
LIN {X 0,Y 573.065,Z 344.313,A -85,B 0,C 180,E1 -2088.91,E2 -2088.91} C_VEL
LIN {X 0,Y 573.072,Z 339.39,A -85,B 0,C 180,E1 -2089.708,E2 -2089.708} C_VEL
LIN {X 0,Y 573.122,Z 332.253,A -85,B 0,C 180,E1 -2090.642,E2 -2090.642} C_VEL
LIN {X 0,Y 573.197,Z 323.93,A -85,B 0,C 180,E1 -2091.486,E2 -2091.486} C_VEL
LIN {X 0,Y 573.245,Z 315.819,A -85,B 0,C 180,E1 -2092.147,E2 -2092.147} C_VEL
LIN {X 0,Y 573.301,Z 308.786,A -85,B 0,C 180,E1 -2092.619,E2 -2092.619} C_VEL
LIN {X 0,Y 573.415,Z 300.109,A -85,B 0,C 180,E1 -2093.091,E2 -2093.091} C_VEL
LIN {X 0,Y 573.441,Z 290.839,A -85,B 0,C 180,E1 -2093.481,E2 -2093.481} C_VEL
LIN {X 0,Y 573.372,Z 282.116,A -85,B 0,C 180,E1 -2093.756,E2 -2093.756} C_VEL
LIN {X 0,Y 572.939,Z 278.728,A -85,B 0,C 180,E1 -2093.854,E2 -2093.854} C_VEL
LIN {X 0,Y 572.943,Z 274.581,A -85,B 0,C 180,E1 -2096.439,E2 -2096.439} C_VEL
LIN {X 0,Y 572.959,Z 269.815,A -85,B 0,C 180,E1 -2099.442,E2 -2099.442} C_VEL
LIN {X 0,Y 572.96,Z 265.519,A -85,B 0,C 180,E1 -2102.186,E2 -2102.186} C_VEL
LIN {X 0,Y 572.945,Z 261.69,A -85,B 0,C 180,E1 -2104.733,E2 -2104.733} C_VEL
LIN {X 0,Y 573.013,Z 257.279,A -85,B 0,C 180,E1 -2107.823,E2 -2107.823} C_VEL
LIN {X 0,Y 573.047,Z 253.379,A -85,B 0,C 180,E1 -2110.54,E2 -2110.54} C_VEL
LIN {X 0,Y 573.123,Z 248.882,A -85,B 0,C 180,E1 -2113.659,E2 -2113.659} C_VEL
LIN {X 0,Y 573.128,Z 246.019,A -85,B 0,C 180,E1 -2115.659,E2 -2115.659} C_VEL
LIN {X 0,Y 573.239,Z 245.892,A -85,B 0,C 180,E1 -2117.602,E2 -2117.602} C_VEL
LIN {X 0,Y 573.233,Z 245.892,A -85,B 0,C 180,E1 -2120.568,E2 -2120.568} C_VEL
LIN {X 0,Y 573.239,Z 245.893,A -85,B 0,C 180,E1 -2123.079,E2 -2123.079} C_VEL
LIN {X 0,Y 573.256,Z 245.893,A -85,B 0,C 180,E1 -2125.673,E2 -2125.673} C_VEL
LIN {X 0,Y 573.221,Z 245.893,A -85,B 0,C 180,E1 -2128.186,E2 -2128.186} C_VEL
LIN {X 0,Y 573.251,Z 245.895,A -85,B 0,C 180,E1 -2130.636,E2 -2130.636} C_VEL
LIN {X 0,Y 573.237,Z 245.891,A -85,B 0,C 180,E1 -2133.025,E2 -2133.025} C_VEL
LIN {X 0,Y 573.255,Z 245.895,A -85,B 0,C 180,E1 -2135.367,E2 -2135.367} C_VEL
LIN {X 0,Y 573.216,Z 245.898,A -85,B 0,C 180,E1 -2138.421,E2 -2138.421} C_VEL
LIN {X 0,Y 573.264,Z 245.888,A -85,B 0,C 180,E1 -2140.729,E2 -2140.729} C_VEL
LIN {X 0,Y 573.233,Z 245.893,A -85,B 0,C 180,E1 -2143.623,E2 -2143.623} C_VEL
LIN {X 0,Y 573.218,Z 245.898,A -85,B 0,C 180,E1 -2146.531,E2 -2146.531} C_VEL
LIN {X 0,Y 573.27,Z 245.886,A -85,B 0,C 180,E1 -2148.735,E2 -2148.735} C_VEL
LIN {X 0,Y 573.241,Z 245.892,A -85,B 0,C 180,E1 -2151.541,E2 -2151.541} C_VEL
LIN {X 0,Y 573.275,Z 245.892,A -85,B 0,C 180,E1 -2154.373,E2 -2154.373} C_VEL
LIN {X 0,Y 573.304,Z 245.884,A -85,B 0,C 180,E1 -2157.191,E2 -2157.191} C_VEL
LIN {X 0,Y 573.302,Z 245.883,A -85,B 0,C 180,E1 -2160.001,E2 -2160.001} C_VEL
LIN {X 0,Y 573.294,Z 245.884,A -85,B 0,C 180,E1 -2162.812,E2 -2162.812} C_VEL
LIN {X 0,Y 573.286,Z 245.888,A -85,B 0,C 180,E1 -2165.629,E2 -2165.629} C_VEL
LIN {X 0,Y 573.278,Z 245.89,A -85,B 0,C 180,E1 -2168.461,E2 -2168.461} C_VEL
LIN {X 0,Y 573.262,Z 245.889,A -85,B 0,C 180,E1 -2171.313,E2 -2171.313} C_VEL
LIN {X 0,Y 573.265,Z 245.887,A -85,B 0,C 180,E1 -2174.194,E2 -2174.194} C_VEL
LIN {X 0,Y 573.248,Z 245.89,A -85,B 0,C 180,E1 -2177.113,E2 -2177.113} C_VEL
LIN {X 0,Y 573.23,Z 245.893,A -85,B 0,C 180,E1 -2180.078,E2 -2180.078} C_VEL
LIN {X 0,Y 573.231,Z 245.892,A -85,B 0,C 180,E1 -2182.339,E2 -2182.339} C_VEL
LIN {X 0,Y 573.241,Z 245.891,A -85,B 0,C 180,E1 -2185.412,E2 -2185.412} C_VEL
LIN {X 0,Y 573.217,Z 245.894,A -85,B 0,C 180,E1 -2188.566,E2 -2188.566} C_VEL
LIN {X 0,Y 573.232,Z 245.896,A -85,B 0,C 180,E1 -2190.994,E2 -2190.994} C_VEL
LIN {X 0,Y 573.256,Z 245.89,A -85,B 0,C 180,E1 -2193.525,E2 -2193.525} C_VEL
LIN {X 0,Y 573.185,Z 245.899,A -85,B 0,C 180,E1 -2196.054,E2 -2196.054} C_VEL
LIN {X 0,Y 573.243,Z 245.897,A -85,B 0,C 180,E1 -2198.702,E2 -2198.702} C_VEL
LIN {X 0,Y 573.226,Z 245.894,A -85,B 0,C 180,E1 -2201.458,E2 -2201.458} C_VEL
LIN {X 0,Y 573.218,Z 245.894,A -85,B 0,C 180,E1 -2204.336,E2 -2204.336} C_VEL
LIN {X 0,Y 573.236,Z 245.892,A -85,B 0,C 180,E1 -2207.36,E2 -2207.36} C_VEL
LIN {X 0,Y 573.27,Z 245.89,A -85,B 0,C 180,E1 -2209.479,E2 -2209.479} C_VEL
LIN {X 0,Y 573.226,Z 245.893,A -85,B 0,C 180,E1 -2212.193,E2 -2212.193} C_VEL
LIN {X 0,Y 573.232,Z 245.893,A -85,B 0,C 180,E1 -2215.23,E2 -2215.23} C_VEL
LIN {X 0,Y 573.323,Z 246.072,A -85,B 0,C 180,E1 -2216.523,E2 -2216.523} C_VEL
LIN {X 0,Y 573.6,Z 249.525,A -85,B 0,C 180,E1 -2217.717,E2 -2217.717} C_VEL
LIN {X 0,Y 573.552,Z 256.127,A -85,B 0,C 180,E1 -2219.843,E2 -2219.843} C_VEL
LIN {X 0,Y 573.431,Z 264.891,A -85,B 0,C 180,E1 -2222.64,E2 -2222.64} C_VEL
LIN {X 0,Y 573.344,Z 273.956,A -85,B 0,C 180,E1 -2225.37,E2 -2225.37} C_VEL
LIN {X 0,Y 573.264,Z 283.094,A -85,B 0,C 180,E1 -2228.044,E2 -2228.044} C_VEL
LIN {X 0,Y 573.174,Z 292.408,A -85,B 0,C 180,E1 -2230.759,E2 -2230.759} C_VEL
LIN {X 0,Y 573.14,Z 302.314,A -85,B 0,C 180,E1 -2233.62,E2 -2233.62} C_VEL
LIN {X 0,Y 573.089,Z 312.533,A -85,B 0,C 180,E1 -2236.527,E2 -2236.527} C_VEL
LIN {X 0,Y 573.072,Z 321.729,A -85,B 0,C 180,E1 -2239.115,E2 -2239.115} C_VEL
LIN {X 0,Y 573.034,Z 325.306,A -85,B 0,C 180,E1 -2240.114,E2 -2240.114} C_VEL
LIN {X 0,Y 573.515,Z 332.451,A -85,B 0,C 180,E1 -2240.301,E2 -2240.301} C_VEL
LIN {X 0,Y 573.44,Z 340.918,A -85,B 0,C 180,E1 -2240.566,E2 -2240.566} C_VEL
LIN {X 0,Y 573.378,Z 349.419,A -85,B 0,C 180,E1 -2240.921,E2 -2240.921} C_VEL
LIN {X 0,Y 573.319,Z 357.747,A -85,B 0,C 180,E1 -2241.364,E2 -2241.364} C_VEL
LIN {X 0,Y 573.272,Z 365.783,A -85,B 0,C 180,E1 -2241.896,E2 -2241.896} C_VEL
LIN {X 0,Y 573.193,Z 374.442,A -85,B 0,C 180,E1 -2242.604,E2 -2242.604} C_VEL
LIN {X 0,Y 573.151,Z 381.592,A -85,B 0,C 180,E1 -2243.327,E2 -2243.327} C_VEL
LIN {X 0,Y 573.113,Z 388.44,A -85,B 0,C 180,E1 -2244.195,E2 -2244.195} C_VEL
LIN {X 0,Y 572.995,Z 393.993,A -85,B 0,C 180,E1 -2245.076,E2 -2245.076} C_VEL
LIN {X 0,Y 573.024,Z 399.152,A -85,B 0,C 180,E1 -2246.133,E2 -2246.133} C_VEL
LIN {X 0,Y 572.99,Z 401.791,A -85,B 0,C 180,E1 -2246.837,E2 -2246.837} C_VEL
LIN {X 0,Y 572.94,Z 404.684,A -85,B 0,C 180,E1 -2247.892,E2 -2247.892} C_VEL
LIN {X 0,Y 572.944,Z 405.936,A -85,B 0,C 180,E1 -2248.595,E2 -2248.595} C_VEL
LIN {X 0,Y 572.937,Z 406.71,A -85,B 0,C 180,E1 -2249.298,E2 -2249.298} C_VEL
LIN {X 0,Y 572.935,Z 407,A -85,B 0,C 180,E1 -2250.001,E2 -2250.001} C_VEL
LIN {X 0,Y 572.937,Z 406.709,A -85,B 0,C 180,E1 -2250.704,E2 -2250.704} C_VEL
LIN {X 0,Y 572.944,Z 405.933,A -85,B 0,C 180,E1 -2251.407,E2 -2251.407} C_VEL
LIN {X 0,Y 572.94,Z 404.679,A -85,B 0,C 180,E1 -2252.11,E2 -2252.11} C_VEL
LIN {X 0,Y 572.99,Z 401.785,A -85,B 0,C 180,E1 -2253.165,E2 -2253.165} C_VEL
LIN {X 0,Y 573.024,Z 399.144,A -85,B 0,C 180,E1 -2253.869,E2 -2253.869} C_VEL
LIN {X 0,Y 572.995,Z 393.981,A -85,B 0,C 180,E1 -2254.926,E2 -2254.926} C_VEL
LIN {X 0,Y 573.138,Z 387.18,A -85,B 0,C 180,E1 -2255.984,E2 -2255.984} C_VEL
LIN {X 0,Y 573.165,Z 379.8,A -85,B 0,C 180,E1 -2256.86,E2 -2256.86} C_VEL
LIN {X 0,Y 573.218,Z 372.396,A -85,B 0,C 180,E1 -2257.575,E2 -2257.575} C_VEL
LIN {X 0,Y 573.303,Z 364.532,A -85,B 0,C 180,E1 -2258.194,E2 -2258.194} C_VEL
LIN {X 0,Y 573.383,Z 354.716,A -85,B 0,C 180,E1 -2258.814,E2 -2258.814} C_VEL
LIN {X 0,Y 573.441,Z 343.28,A -85,B 0,C 180,E1 -2259.346,E2 -2259.346} C_VEL
LIN {X 0,Y 573.521,Z 333.215,A -85,B 0,C 180,E1 -2259.679,E2 -2259.679} C_VEL
LIN {X 0,Y 573.228,Z 326.987,A -85,B 0,C 180,E1 -2259.84,E2 -2259.84} C_VEL
LIN {X 0,Y 573.034,Z 325.299,A -85,B 0,C 180,E1 -2259.888,E2 -2259.888} C_VEL
LIN {X 0,Y 573.08,Z 316.358,A -85,B 0,C 180,E1 -2262.394,E2 -2262.394} C_VEL
LIN {X 0,Y 573.137,Z 306.139,A -85,B 0,C 180,E1 -2265.287,E2 -2265.287} C_VEL
LIN {X 0,Y 573.183,Z 295.921,A -85,B 0,C 180,E1 -2268.221,E2 -2268.221} C_VEL
LIN {X 0,Y 573.261,Z 285.37,A -85,B 0,C 180,E1 -2271.293,E2 -2271.293} C_VEL
LIN {X 0,Y 573.306,Z 275.297,A -85,B 0,C 180,E1 -2274.247,E2 -2274.247} C_VEL
LIN {X 0,Y 573.435,Z 266.195,A -85,B 0,C 180,E1 -2276.967,E2 -2276.967} C_VEL
LIN {X 0,Y 573.509,Z 258.045,A -85,B 0,C 180,E1 -2279.534,E2 -2279.534} C_VEL
LIN {X 0,Y 573.59,Z 251.052,A -85,B 0,C 180,E1 -2281.795,E2 -2281.795} C_VEL
LIN {X 0,Y 573.495,Z 247.296,A -85,B 0,C 180,E1 -2283.048,E2 -2283.048} C_VEL
LIN {X 0,Y 573.286,Z 245.891,A -85,B 0,C 180,E1 -2283.576,E2 -2283.576} C_VEL
LIN {X 0,Y 573.259,Z 245.892,A -85,B 0,C 180,E1 -2286.923,E2 -2286.923} C_VEL
LIN {X 0,Y 573.246,Z 245.894,A -85,B 0,C 180,E1 -2289.608,E2 -2289.608} C_VEL
